// SIMATIC STEP 7 (V5.x) project DAYSILAUTOCLAVE
// CPU: CPU 315-2 PN/DP
// station: Hardware
// station: SLIO_CPU_015
// station: P_ADR_BUS
// program: S7 Program(1)
// program: 271220024

SYMBOL_TABLE
"AI-SENSOR-DATA"	DB 1	DB 1
"ORTAK_DATA"	DB 2	DB 2	// Ortak Veriler
"TIME_OTO_1_DB"	DB 5	SFB 4
"TIME_OTO_2_DB"	DB 6	SFB 4
"TIME_OTO_1_PROSES_DB"	DB 7	SFB 4
"TIME_OTO_2_PROSES_DB"	DB 8	SFB 4
"SURELER_DB"	DB 14	FB 3
"SAFETY_DB"	DB 15	FB 2
"KAZAN1_DATA"	DB 17	DB 17
"KAZAN2_DATA"	DB 18	DB 18	// KAZAN 2 BILGILERI
"JEN1_DATA"	DB 19	DB 19
"JEN2_DATA"	DB 20	DB 20
"JEN1_PID_DATA"	DB 21	DB 21
"JEN2_PID_DATA"	DB 22	DB 22
"KAZAN1_PID_DATA"	DB 23	DB 23	// KAZAN 1 PID BILGILERI
"KAZAN2_PID_DATA"	DB 24	DB 24	// KAZAN 2 PID BILGILERI
"JEN2_KONTROL_BLOGU_DB"	DB 51	FB 50
"JEN_1_PID_DB"	DB 69	FB 58
"JEN_2_PID_DB"	DB 70	FB 58
"OTOKLAV_1_DB"	DB 94	FB 94
"OTOKLAV_2_DB"	DB 95	FB 95
"FB98_DB"	DB 98	FB 98
"FB99_DB"	DB 99	FB 99
"HMI_DATA"	DB 100	DB 100	// Hmi arayuz verileri
"KAZAN_1_PID_DB"	DB 130	FB 58
"KAZAN_2_PID_DATA"	DB 231	FB 58
"MAINBLOCK"	FB 1	FB 1	// ANA PROGRAM BLOGU
"SAFETY"	FB 2	FB 2
"SURELER"	FB 3	FB 3
"TEST_BLOGU"	FB 5	FB 5
"KAZAN_ORTAK"	FB 20	FB 20
"KAZAN_PID_ORTAK"	FB 21	FB 21
"CONT_C"	FB 41	FB 41	// Continuous Control
"KAZAN_1_PID_KONTROL"	FB 47	FB 47
"KAZAN_2_PID_KONTROL"	FB 48	FB 48
"JEN1_PID_KONTROL"	FB 49	FB 49
"JEN2_PID_KONTROL"	FB 50	FB 50	// BUAHR JENERATÖR 2 PID
"TCONT_CP"	FB 58	FB 58	// temperature PID controller with pulse generator and self-tuning
"KAZAN_1_KONTROL"	FB 94	FB 94
"KAZAN_2_KONTROL"	FB 95	FB 95
"KAZAN1_KONTROL_BLOGU"	FB 96	FB 96
"KAZAN2_KONTROL_BLOGU"	FB 97	FB 97
"JEN1_KONTROL_BLOGU"	FB 98	FB 98
"JEN2_KONTROL_BLOGU"	FB 99	FB 99
"TIME_UNSCALE"	FC 1	FC 1
"S5TI_TIM"	FC 33	FC 33	// S5 Time to IEC Time
"SCALE"	FC 105	FC 105	// Scaling Values
"UNSCALE"	FC 106	FC 106	// Unscaling Values
"KAZAN1_ACIL_STOP"	I 0.0	BOOL	// Acil Stop
"KAZAN1_START"	I 0.1	BOOL	// Kazan 1 Start
"KAZAN1_TRANSFER"	I 0.2	BOOL	// Kazan 1 Buhar Transferi
"KAZAN1_BOSALTIM"	I 0.3	BOOL	// Kazan 1 Bosaltim
"KAZAN1_KAPAK_SW"	I 0.4	BOOL	// Kazan 1 Kapak Kapandi
"KAZAN2_ACIL_STOP"	I 0.5	BOOL	// Kazan 2 Acil Stop
"KAZAN2_START"	I 0.6	BOOL	// Kazan 2 Start
"KAZAN2_TRANSFER"	I 0.7	BOOL	// Kazan 2 Buhar Transferi
"KAZAN2_BOSALTIM"	I 1.0	BOOL	// Kazan 2 Bosaltim
"KAZAN2_KAPAK_SW"	I 1.1	BOOL	// Kazan 2 Kapak Kapandi
"JEN1_STOP"	I 1.2	BOOL	// Jenerator 1 Stop
"JEN1_START"	I 1.3	BOOL	// Jenerator 1 Start
"JEN2_STOP"	I 1.4	BOOL	// Jenerator 2 Stop
"JEN2_START"	I 1.5	BOOL	// Jenerator 2 Start
"MANUEL"	I 1.6	BOOL	// Manuel Mod
"OTOMATIK"	I 1.7	BOOL	// Otomatik Mod
"JEN2_MOTOR_CALISTI"	I 2.0	BOOL
"JEN_1_MIN_SU_SEVIYESI"	I 3.0	BOOL
"JEN_2_MIN_SU_SEVIYESI"	I 3.1	BOOL
"0.1 SN."	M 0.0	BOOL
"0.2 SN."	M 0.1	BOOL
"0.4 SN."	M 0.2	BOOL
"0.5 SN."	M 0.3	BOOL
"0.8 SN."	M 0.4	BOOL
"1.0 SN."	M 0.5	BOOL
"1.6 SN."	M 0.6	BOOL
"2.0 SN."	M 0.7	BOOL
"Oto_1_Proses_BASLADI"	M 20.0	BOOL
"Oto_2_Proses_Basladi"	M 20.1	BOOL
"JEN2_CALIS_SURESI_BASLA"	M 22.0	BOOL
"JEN2_CALISTI_RIS"	M 22.1	BOOL
"JEN1_CALIS_SURESI_BASLA"	M 23.0	BOOL
"JEN1_CALISTI_RIS"	M 23.1	BOOL
"Jen1_Guvenlik_set_reset"	M 25.0	BOOL
"Jen2_Guvenlik_Set_Reset"	M 26.0	BOOL
"OTO_1_BEKLEME_BASLADI"	M 27.0	BOOL
"OTO_2_BEKLEME_BASLADI"	M 27.1	BOOL
"KAZAN_1_PID_MAN_ON"	M 35.0	BOOL
"KAZAN_2_MAN_ON"	M 37.0	BOOL
"TEST_START"	M 40.0	BOOL
"TEST_STOP"	M 40.1	BOOL
"TEST_OUT"	M 40.2	BOOL
"ALWAYS OFF"	M 100.0	BOOL	// ALWAYS OFF
"ALWAYS ON"	M 100.1	BOOL	// ALWAYS ON
"SET2_ULASMADI_SR"	M 101.0	BOOL
"SET2_ULASMADI_RIS"	M 101.1	BOOL
"JEN2_TCONT_MAN_ON"	M 155.0	BOOL
"Jen2_Stop_Trigger"	M 200.0	BOOL
"Jen2_Stop_Ris"	M 200.1	BOOL
"Jen2_Stop_Set_Mem"	M 200.2	BOOL
"JEN2_STOP_SET_RESET"	M 201.0	BOOL
"Sicaklik Dustu"	M 201.1	BOOL
"Ris_Jen2_Sicaklik_Dustu"	M 201.2	BOOL
"Rising_Sogutma"	M 201.3	BOOL
"Falling_Sogutma"	M 201.4	BOOL
"JEN1_STOP_SET_RESET"	M 202.0	BOOL
"START"	M 700.1	BOOL
"PID_START"	M 700.2	BOOL
"BRULOR_START"	M 700.3	BOOL
"SICAKLIK_1_OK"	M 700.5	BOOL
"SICAKLIK_2_OK"	M 700.6	BOOL
"BURLOR_MOTOR_START"	M 700.7	BOOL
"STOP"	M 701.1	BOOL
"100_DERECE_RIS"	M 750.0	BOOL
"Jen2_Ris"	M 750.4	BOOL
"Jen1_Ris"	M 750.5	BOOL
"BOS"	M 1000.0	BOOL
"PID BLOCK"	OB 35	OB 35	// PID BLOCK
"ZAMANHATASI"	OB 80	OB 80	// ZAMAN HATASI
"GERILIMHATASI"	OB 81	OB 81	// BESLEME GERILIMI HATASI
"HATAUYARISI"	OB 82	OB 82	// HATA UYARISI
"TAKMACIKARMAHATASI"	OB 83	OB 83	// TAKMA ÇIKARMA UYARISI
"CPUHARDWAREERROR"	OB 84	OB 84	// CPU HARDWARE ERROR
"PROGRAMHATASI"	OB 85	OB 85	// PROGRAM YURUTME HATASI
"RACKHATASI"	OB 86	OB 86	// RACK HATASI
"HABERLESMEHATASI"	OB 87	OB 87	// HABERLESME HATASI,
"COMPLETE RESTART"	OB 100	OB 100	// Complete Restart
"RESTART"	OB 101	OB 101	// Restart
"COLD RESTART"	OB 102	OB 102	// Cold Restart
"PROGRAMMINGERROR"	OB 121	OB 121	// PROGRAMLAMA HATASI
"KAZAN1_YESIL_LAMBA"	Q 0.0	BOOL	// Kazan 1 Yesil Lamba
"KAZAN1_KIRMIZI_LAMBA"	Q 0.1	BOOL	// Kazan 1 Kirmizi Lamba
"KAZAN1_DUDUK"	Q 0.2	BOOL	// Kazan 1 Duduk
"KAZAN1_BOSALTIM_VALFI"	Q 0.3	BOOL	// Kazan 1 Buhar Bosaltim
"KAZAN1_TRANS_BUT_LAMBASI"	Q 0.4	BOOL	// Kazan 1 Transfer Lambasi
"KAZAN1_EMN_VALFI_BOS"	Q 0.5	BOOL	// Kazan  1 Emniyet vantili bosaltim valfi
"KAZAN2_YESIL_LAMBA"	Q 0.6	BOOL	// Kazan 2 Yesil Lamba
"KAZAN2_KIRMIZI_LAMBA"	Q 0.7	BOOL	// Kazan 2 Kirmizi Lamba
"KAZAN2_DUDUK"	Q 1.0	BOOL	// Kazan 2 Duduk
"KAZAN2_BOSALTIM_VALFI"	Q 1.1	BOOL	// Kazan 2 Buhar Bosaltim
"KAZAN2_TRANS_BUT_LAMBASI"	Q 1.2	BOOL	// Kazan 2 Transfer Lambasi
"KAZAN2_EMN_VALFI_BOS"	Q 1.3	BOOL	// Kazan Emniyet vantili bosaltim valfi
"JEN_1_HAT_VANASI"	Q 1.4	BOOL
"JEN_1_PANO_STOP_LAMBASI"	Q 1.5	BOOL
"JEN_1_PANO_START_LAMBASI"	Q 1.6	BOOL
"JEN_2_HAT_VANASI"	Q 1.7	BOOL
"JEN_2_PANO_STOP_LAMBASI"	Q 2.0	BOOL
"JEN_2_PANO_START_LAMBASI"	Q 2.1	BOOL
"PANO_OTO_MAN_BUTON_LAMBA"	Q 2.2	BOOL
"PANO_ALARM"	Q 2.3	BOOL
"JEN_1_BRULOR"	Q 2.4	BOOL
"JEN_1_POMPA"	Q 2.5	BOOL
"JEN_2_BRULOR_OUT"	Q 2.6	BOOL
"JEN_2_SU_POM_OUT"	Q 2.7	BOOL
"TON"	SFB 4	SFB 4	// Generate an On Delay
"delay_300ms_1"	T 8	TIMER
"500ms_delay1"	T 10	TIMER
"1s Delay"	T 11	TIMER
"Pisim_Suresi"	T 12	TIMER
"500ms_delay"	T 13	TIMER
"s_offt_7s_delay"	T 14	TIMER
"tm_adim1_pid_basla_delay"	T 16	TIMER
"500ms_delay_kazan_2"	T 20	TIMER
"1ms_delay_kazan_2"	T 21	TIMER
"kazan_2_pisirme_delay"	T 22	TIMER
"kazan_2_500ms_delay"	T 23	TIMER
"kazan_2_7s_delay"	T 24	TIMER
"Delay_500ms_Jen2"	T 30	TIMER
"DELAY_1S_JEN_HATA"	T 33	TIMER
"DELAY_300MS"	T 42	TIMER
"DELAY_500MS_1"	T 43	TIMER
"DELAY_5S_pompa"	T 44	TIMER
"OTO_2_DELAY_BITIS"	T 50	TIMER
"OTO_1_DELAY_PISIM_BITTI"	T 51	TIMER
"DELAY_ADIM5_BEKLE"	T 52	TIMER
"DELAY_ADIM5_BEKLE2"	T 53	TIMER
"TIM_SET2_ULASMADI"	T 57	TIMER
"TEST BLOGU VAT"	VAT 1	
"JEN2_MONITOR"	VAT 2	
"KAZAN-1-MONITOR"	VAT 3	
"KAZAN-2-MONITOR"	VAT 4	
"JEN1_MONITOR"	VAT 5	
"deneme"	VAT 6	
END_SYMBOL_TABLE

FUNCTION_BLOCK "MAINBLOCK"	// FB 1
VERSION : 0.1
BEGIN
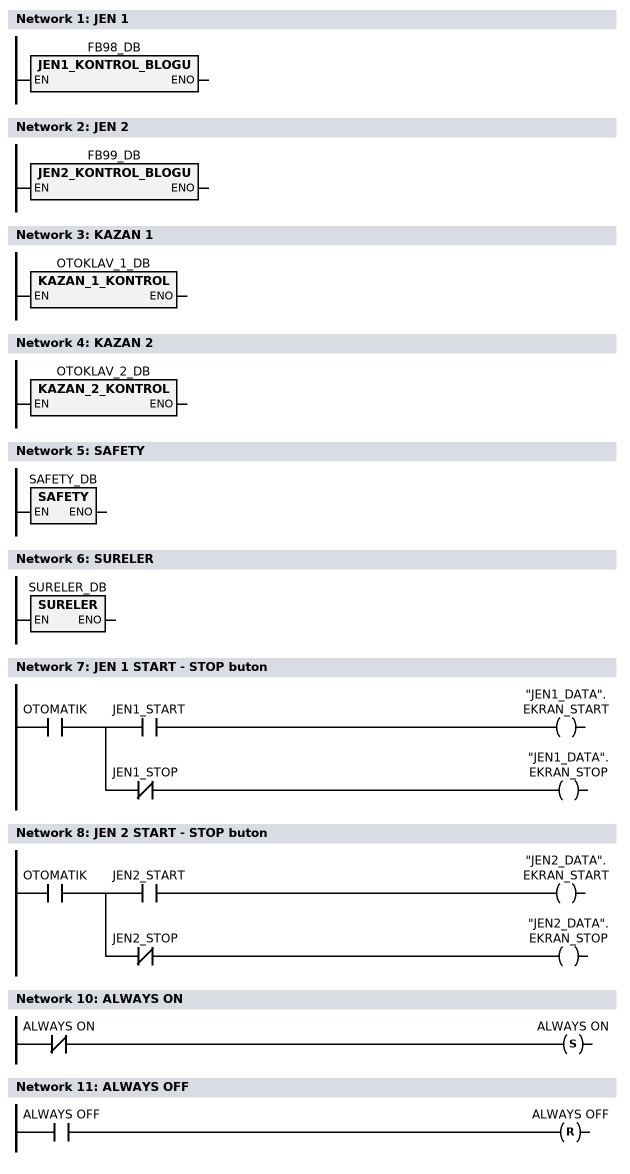
NETWORK
TITLE = JEN 1
      CALL  "JEN1_KONTROL_BLOGU" , "FB98_DB";
      NOP   0;
NETWORK
TITLE = JEN 2
      CALL  "JEN2_KONTROL_BLOGU" , "FB99_DB";
      NOP   0;
NETWORK
TITLE = KAZAN 1
      CALL  "KAZAN_1_KONTROL" , "OTOKLAV_1_DB";
      NOP   0;
NETWORK
TITLE = KAZAN 2
      CALL  "KAZAN_2_KONTROL" , "OTOKLAV_2_DB";
      NOP   0;
NETWORK
TITLE = SAFETY
      CALL  "SAFETY" , "SAFETY_DB";
      NOP   0;
NETWORK
TITLE = SURELER
      CALL  "SURELER" , "SURELER_DB";
      NOP   0;
NETWORK
TITLE = JEN 1 START - STOP buton
      A     "OTOMATIK";
      =     L 0.0;
      A     L 0.0;
      A     "JEN1_START";
      =     "JEN1_DATA".EKRAN_START;
      A     L 0.0;
      AN    "JEN1_STOP";
      =     "JEN1_DATA".EKRAN_STOP;
NETWORK
TITLE = JEN 2 START - STOP buton
      A     "OTOMATIK";
      =     L 0.0;
      A     L 0.0;
      A     "JEN2_START";
      =     "JEN2_DATA".EKRAN_START;
      A     L 0.0;
      AN    "JEN2_STOP";
      =     "JEN2_DATA".EKRAN_STOP;
NETWORK
TITLE =
NETWORK
TITLE = ALWAYS ON
      AN    "ALWAYS ON";
      S     "ALWAYS ON";
NETWORK
TITLE = ALWAYS OFF
      A     "ALWAYS OFF";
      R     "ALWAYS OFF";
NETWORK
TITLE =
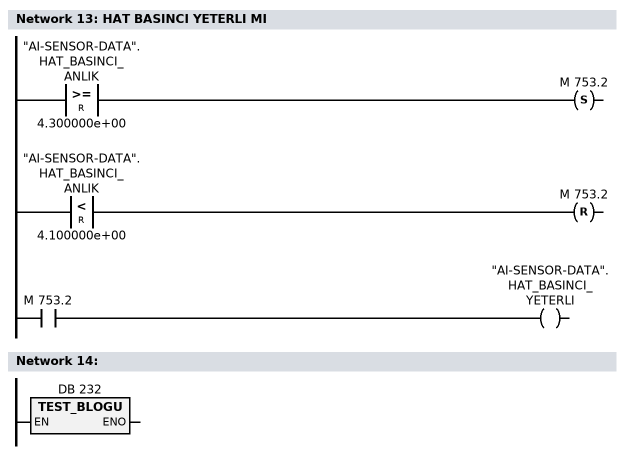
NETWORK
TITLE = HAT BASINCI YETERLI MI
      A(;
      L     "AI-SENSOR-DATA".HAT_BASINCI_ANLIK;
      L     4.300000e+00;
      >=R;
      );
      S     M 753.2;
      A(;
      L     "AI-SENSOR-DATA".HAT_BASINCI_ANLIK;
      L     4.100000e+00;
      <R;
      );
      R     M 753.2;
      A     M 753.2;
      =     "AI-SENSOR-DATA".HAT_BASINCI_YETERLI;
NETWORK
TITLE =
      CALL  "TEST_BLOGU" , DB 232;
      NOP   0;
END_FUNCTION_BLOCK

FUNCTION_BLOCK "SAFETY"	// FB 2
VERSION : 0.1
BEGIN
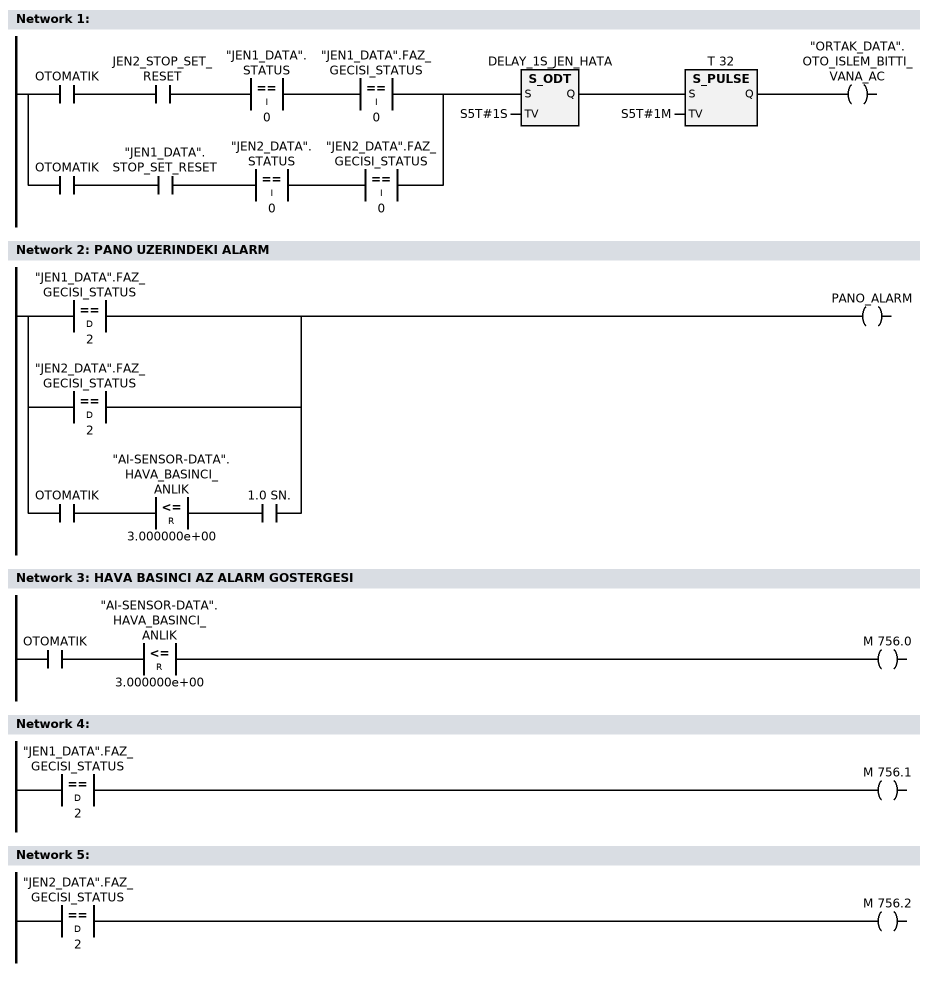
NETWORK
TITLE =
      A(;
      A(;
      A     "OTOMATIK";
      A     "JEN2_STOP_SET_RESET";
      A(;
      L     "JEN1_DATA".STATUS;
      L     0;
      ==I;
      );
      A(;
      L     "JEN1_DATA".FAZ_GECISI_STATUS;
      L     0;
      ==I;
      );
      O;
      A     "OTOMATIK";
      A     "JEN1_DATA".STOP_SET_RESET;
      A(;
      L     "JEN2_DATA".STATUS;
      L     0;
      ==I;
      );
      A(;
      L     "JEN2_DATA".FAZ_GECISI_STATUS;
      L     0;
      ==I;
      );
      );
      L     S5T#1S;
      SD    "DELAY_1S_JEN_HATA";
      NOP   0;
      NOP   0;
      NOP   0;
      A     "DELAY_1S_JEN_HATA";
      );
      L     S5T#1M;
      SP    T 32;
      NOP   0;
      NOP   0;
      NOP   0;
      A     T 32;
      =     "ORTAK_DATA".OTO_ISLEM_BITTI_VANA_AC;
NETWORK
TITLE = PANO UZERINDEKI ALARM 
//JENERATORDE MINIMUM SU SEVIYESINE DUSERSE PANO UZERINDEKI ALARMI CALISTIR
      O(;
      L     "JEN1_DATA".FAZ_GECISI_STATUS;
      L     2;
      ==D;
      );
      O(;
      L     "JEN2_DATA".FAZ_GECISI_STATUS;
      L     2;
      ==D;
      );
      O;
      A     "OTOMATIK";
      A(;
      L     "AI-SENSOR-DATA".HAVA_BASINCI_ANLIK;
      L     3.000000e+00;
      <=R;
      );
      A     "1.0 SN.";
      =     "PANO_ALARM";
NETWORK
TITLE = HAVA BASINCI AZ ALARM GOSTERGESI
      A     "OTOMATIK";
      A(;
      L     "AI-SENSOR-DATA".HAVA_BASINCI_ANLIK;
      L     3.000000e+00;
      <=R;
      );
      =     M 756.0;
NETWORK
TITLE =
      L     "JEN1_DATA".FAZ_GECISI_STATUS;
      L     2;
      ==D;
      =     M 756.1;
NETWORK
TITLE =
      L     "JEN2_DATA".FAZ_GECISI_STATUS;
      L     2;
      ==D;
      =     M 756.2;
END_FUNCTION_BLOCK

FUNCTION_BLOCK "SURELER"	// FB 3
VERSION : 0.1
BEGIN
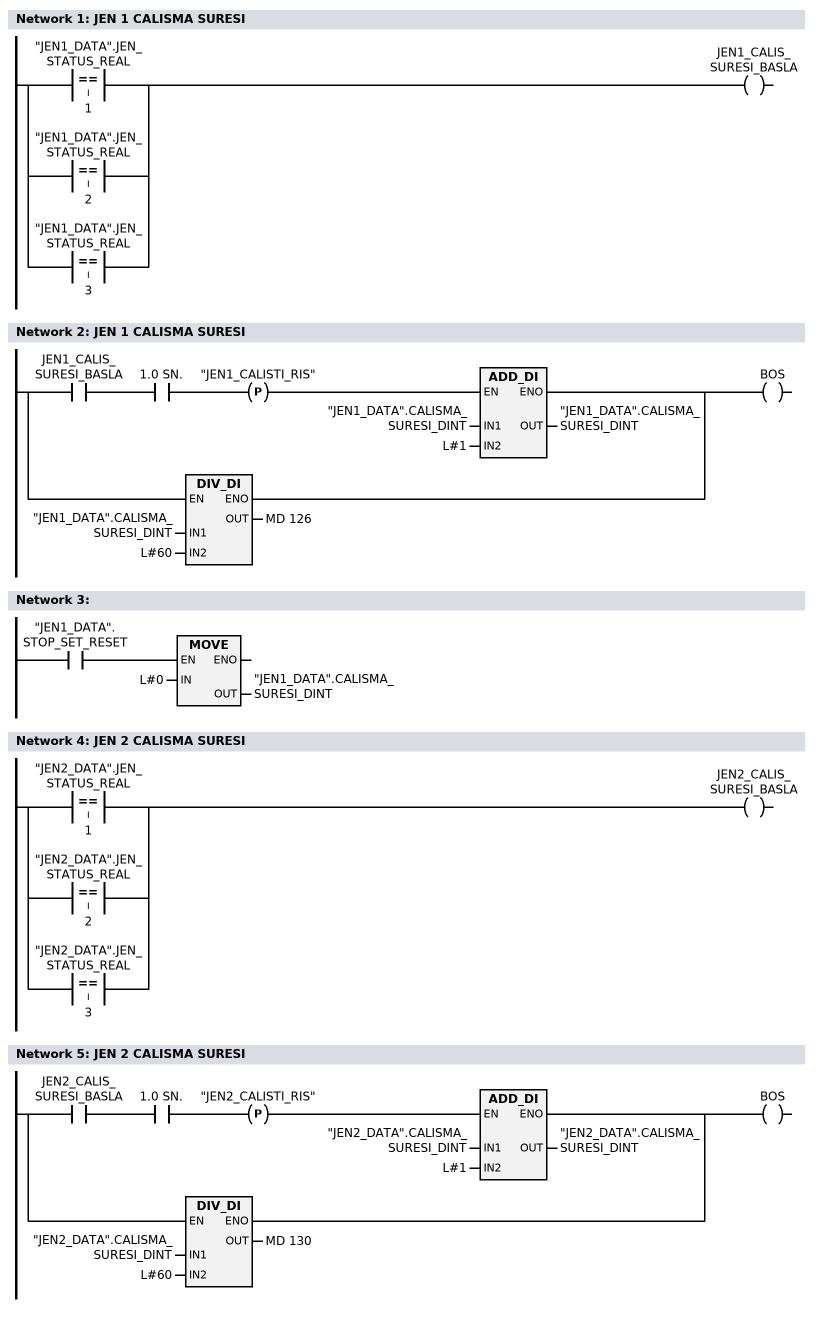
NETWORK
TITLE = JEN 1 CALISMA SURESI
      O(;
      L     "JEN1_DATA".JEN_STATUS_REAL;
      L     1;
      ==I;
      );
      O(;
      L     "JEN1_DATA".JEN_STATUS_REAL;
      L     2;
      ==I;
      );
      O(;
      L     "JEN1_DATA".JEN_STATUS_REAL;
      L     3;
      ==I;
      );
      =     "JEN1_CALIS_SURESI_BASLA";
NETWORK
TITLE = JEN 1 CALISMA SURESI
      O(;
      A     "JEN1_CALIS_SURESI_BASLA";
      A     "1.0 SN.";
      FP    "JEN1_CALISTI_RIS";
      JNB   _001;
      L     "JEN1_DATA".CALISMA_SURESI_DINT;
      L     L#1;
      +D;
      T     "JEN1_DATA".CALISMA_SURESI_DINT;
      AN    OV;
      SAVE;
      CLR;
_001: A     BR;
      );
      O(;
      L     "JEN1_DATA".CALISMA_SURESI_DINT;
      L     L#60;
      /D;
      T     MD 126;
      AN    OV;
      SAVE;
      CLR;
      A     BR;
      );
      =     "BOS";
NETWORK
TITLE =
      A     "JEN1_DATA".STOP_SET_RESET;
      JNB   _002;
      L     L#0;
      T     "JEN1_DATA".CALISMA_SURESI_DINT;
_002: NOP   0;
NETWORK
TITLE = JEN 2 CALISMA SURESI
      O(;
      L     "JEN2_DATA".JEN_STATUS_REAL;
      L     1;
      ==I;
      );
      O(;
      L     "JEN2_DATA".JEN_STATUS_REAL;
      L     2;
      ==I;
      );
      O(;
      L     "JEN2_DATA".JEN_STATUS_REAL;
      L     3;
      ==I;
      );
      =     "JEN2_CALIS_SURESI_BASLA";
NETWORK
TITLE = JEN 2 CALISMA SURESI
      O(;
      A     "JEN2_CALIS_SURESI_BASLA";
      A     "1.0 SN.";
      FP    "JEN2_CALISTI_RIS";
      JNB   _003;
      L     "JEN2_DATA".CALISMA_SURESI_DINT;
      L     L#1;
      +D;
      T     "JEN2_DATA".CALISMA_SURESI_DINT;
      AN    OV;
      SAVE;
      CLR;
_003: A     BR;
      );
      O(;
      L     "JEN2_DATA".CALISMA_SURESI_DINT;
      L     L#60;
      /D;
      T     MD 130;
      AN    OV;
      SAVE;
      CLR;
      A     BR;
      );
      =     "BOS";
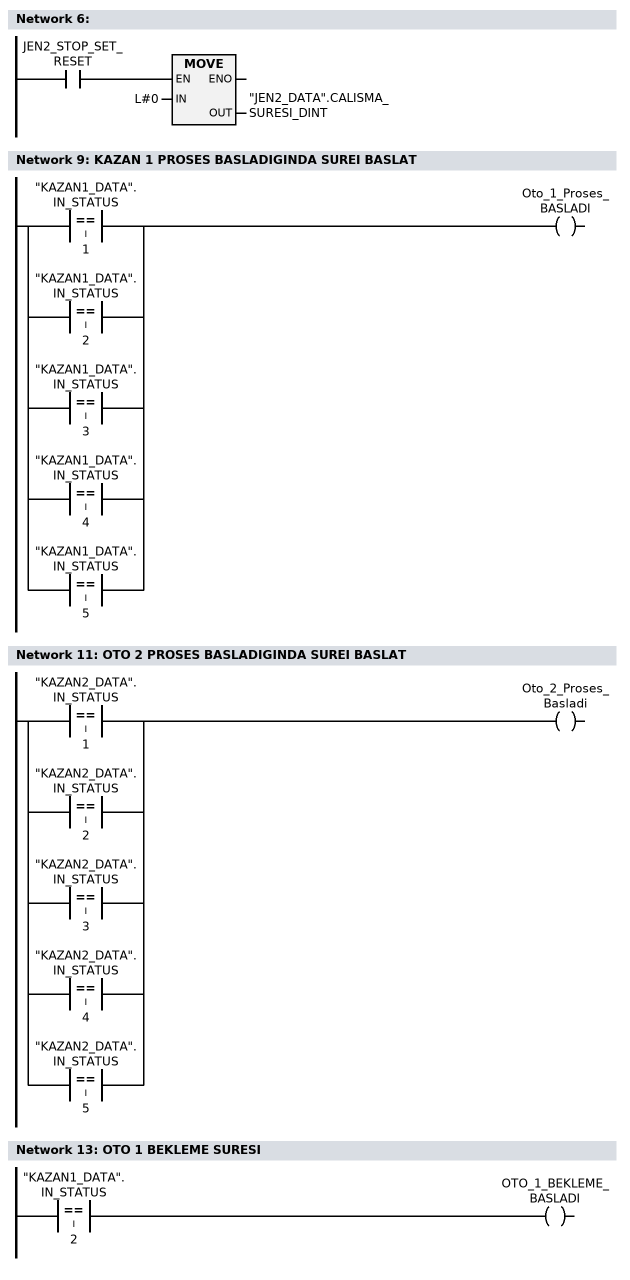
NETWORK
TITLE =
      A     "JEN2_STOP_SET_RESET";
      JNB   _004;
      L     L#0;
      T     "JEN2_DATA".CALISMA_SURESI_DINT;
_004: NOP   0;
NETWORK
TITLE = OTOKLAV 1 PISIM GECEN SURE
      O(;
      A(;
      A     "KAZAN1_DATA".O_PISIM_BASLADI;
      =     L 0.0;
      BLD   103;
      BLD   9;
      =     L 5.0;
      CDB;
      OPN   DI 5;
      TAR2  LD 1;
      A     L 0.0;
      =     DIX 0.0;
      L     L#82800000;
      T     DID 2;
      LAR2  P#DBX 0.0;
      UC    "TON";
      LAR2  LD 1;
      L     DID 8;
      OPN   DI 17;
      T     DID 42;
      OPN   DI 5;
      CDB;
      BLD   10;
      A     BR;
      );
      JNB   _005;
      CALL  "TIME_UNSCALE" (
           iTimeET                  := "KAZAN1_DATA".PISIM_GECEN_SURE_TIME,
           iIstenileSure            := "KAZAN1_DATA".IN_PISIM_SURESI,
           oOUT                     := "KAZAN1_DATA".PISIM_GECEN_SURE_DINT);
_005: A     BR;
      );
      O(;
      L     "KAZAN1_DATA".PISIM_GECEN_SURE_DINT;
      L     60;
      /D;
      T     MD 118;
      AN    OV;
      SAVE;
      CLR;
      A     BR;
      );
      =     "BOS";
NETWORK
TITLE = OTOKLAV 2 PISIM GECEN SURE
      O(;
      A(;
      A     "KAZAN2_DATA".O_PISIM_BASLADI;
      =     L 0.0;
      BLD   103;
      BLD   9;
      =     L 5.0;
      CDB;
      OPN   DI 6;
      TAR2  LD 1;
      A     L 0.0;
      =     DIX 0.0;
      L     L#82800000;
      T     DID 2;
      LAR2  P#DBX 0.0;
      UC    "TON";
      LAR2  LD 1;
      L     DID 8;
      OPN   DI 18;
      T     DID 42;
      OPN   DI 6;
      CDB;
      BLD   10;
      A     BR;
      );
      JNB   _006;
      CALL  "TIME_UNSCALE" (
           iTimeET                  := "KAZAN2_DATA".PISIM_GECEN_SURE_TIME,
           iIstenileSure            := "KAZAN2_DATA".IN_PISIM_SURESI,
           oOUT                     := "KAZAN2_DATA".PISIM_GECEN_SURE_DINT);
_006: A     BR;
      );
      O(;
      L     "KAZAN2_DATA".PISIM_GECEN_SURE_DINT;
      L     60;
      /D;
      T     MD 122;
      AN    OV;
      SAVE;
      CLR;
      A     BR;
      );
      =     "BOS";
NETWORK
TITLE = KAZAN 1 PROSES BASLADIGINDA SUREI BASLAT
      O(;
      L     "KAZAN1_DATA".IN_STATUS;
      L     1;
      ==I;
      );
      O(;
      L     "KAZAN1_DATA".IN_STATUS;
      L     2;
      ==I;
      );
      O(;
      L     "KAZAN1_DATA".IN_STATUS;
      L     3;
      ==I;
      );
      O(;
      L     "KAZAN1_DATA".IN_STATUS;
      L     4;
      ==I;
      );
      O(;
      L     "KAZAN1_DATA".IN_STATUS;
      L     5;
      ==I;
      );
      =     "Oto_1_Proses_BASLADI";
NETWORK
TITLE = OTOKLAV 1 PROSES SURESI
      O(;
      A(;
      A     "Oto_1_Proses_BASLADI";
      =     L 0.0;
      BLD   103;
      BLD   9;
      =     L 5.0;
      CDB;
      OPN   DI 7;
      TAR2  LD 1;
      A     L 0.0;
      =     DIX 0.0;
      L     L#82800000;
      T     DID 2;
      LAR2  P#DBX 0.0;
      UC    "TON";
      LAR2  LD 1;
      L     DID 8;
      OPN   DI 17;
      T     DID 50;
      OPN   DI 7;
      CDB;
      BLD   10;
      A     BR;
      );
      JNB   _007;
      L     "KAZAN1_DATA".PROSES_SURESI_TIME;
      L     1000;
      /D;
      T     "KAZAN1_DATA".PROSES_SURESI_DINT;
      AN    OV;
      SAVE;
      CLR;
_007: A     BR;
      );
      O(;
      L     "KAZAN1_DATA".PROSES_SURESI_DINT;
      L     60;
      /D;
      T     MD 110;
      AN    OV;
      SAVE;
      CLR;
      A     BR;
      );
      =     "BOS";
NETWORK
TITLE = OTO 2 PROSES BASLADIGINDA SUREI BASLAT
      O(;
      L     "KAZAN2_DATA".IN_STATUS;
      L     1;
      ==I;
      );
      O(;
      L     "KAZAN2_DATA".IN_STATUS;
      L     2;
      ==I;
      );
      O(;
      L     "KAZAN2_DATA".IN_STATUS;
      L     3;
      ==I;
      );
      O(;
      L     "KAZAN2_DATA".IN_STATUS;
      L     4;
      ==I;
      );
      O(;
      L     "KAZAN2_DATA".IN_STATUS;
      L     5;
      ==I;
      );
      =     "Oto_2_Proses_Basladi";
NETWORK
TITLE = OTO 2 PROSES_SURESI
      O(;
      A(;
      A     "Oto_2_Proses_Basladi";
      =     L 0.0;
      BLD   103;
      BLD   9;
      =     L 5.0;
      CDB;
      OPN   DI 8;
      TAR2  LD 1;
      A     L 0.0;
      =     DIX 0.0;
      L     L#82800000;
      T     DID 2;
      LAR2  P#DBX 0.0;
      UC    "TON";
      LAR2  LD 1;
      L     DID 8;
      OPN   DI 18;
      T     DID 50;
      OPN   DI 8;
      CDB;
      BLD   10;
      A     BR;
      );
      JNB   _008;
      L     "KAZAN2_DATA".PROSES_SURESI_TIM;
      L     1000;
      /D;
      T     "KAZAN2_DATA".PROSES_SURESI_DINT;
      AN    OV;
      SAVE;
      CLR;
_008: A     BR;
      );
      O(;
      L     "KAZAN2_DATA".PROSES_SURESI_DINT;
      L     60;
      /D;
      T     MD 114;
      AN    OV;
      SAVE;
      CLR;
      A     BR;
      );
      =     "BOS";
NETWORK
TITLE = OTO 1 BEKLEME SURESI
      L     "KAZAN1_DATA".IN_STATUS;
      L     2;
      ==I;
      =     "OTO_1_BEKLEME_BASLADI";
NETWORK
TITLE = OTO 1 BEKLEME SURESI
      A(;
      A     "OTO_1_BEKLEME_BASLADI";
      =     L 0.0;
      BLD   103;
      BLD   9;
      =     L 5.0;
      CDB;
      OPN   DI 9;
      TAR2  LD 1;
      A     L 0.0;
      =     DIX 0.0;
      L     L#82800000;
      T     DID 2;
      LAR2  P#DBX 0.0;
      UC    "TON";
      LAR2  LD 1;
      L     DID 8;
      OPN   DI 17;
      T     DID 58;
      OPN   DI 9;
      CDB;
      BLD   10;
      A     BR;
      );
      JNB   _009;
      L     "KAZAN1_DATA".BEKLEME_SURESI_TIME;
      L     1000;
      /D;
      T     "KAZAN1_DATA".BEKLEME_SURESI_DINT;
_009: NOP   0;
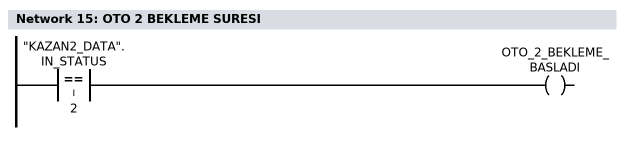
NETWORK
TITLE = OTO 2 BEKLEME SURESI
      L     "KAZAN2_DATA".IN_STATUS;
      L     2;
      ==I;
      =     "OTO_2_BEKLEME_BASLADI";
NETWORK
TITLE = OTO 2 BEKLEME SURESI
      A(;
      A     "OTO_2_BEKLEME_BASLADI";
      =     L 0.0;
      BLD   103;
      BLD   9;
      =     L 5.0;
      CDB;
      OPN   DI 10;
      TAR2  LD 1;
      A     L 0.0;
      =     DIX 0.0;
      L     L#82800000;
      T     DID 2;
      LAR2  P#DBX 0.0;
      UC    "TON";
      LAR2  LD 1;
      L     DID 8;
      OPN   DI 18;
      T     DID 58;
      OPN   DI 10;
      CDB;
      BLD   10;
      A     BR;
      );
      JNB   _00a;
      L     "KAZAN2_DATA".BEKLEME_SURESI_TIME;
      L     1000;
      /D;
      T     "KAZAN2_DATA".BEKLEME_SURESI_DINT;
_00a: NOP   0;
END_FUNCTION_BLOCK

FUNCTION_BLOCK "TEST_BLOGU"	// FB 5
VERSION : 0.1
BEGIN
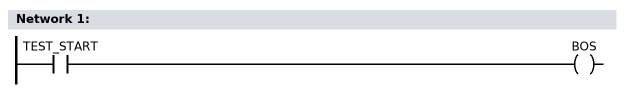
NETWORK
TITLE =
      A     "TEST_START";
      =     "BOS";
END_FUNCTION_BLOCK

FUNCTION_BLOCK "KAZAN_ORTAK"	// FB 20
//0 - baslama kriterleri
//1 - pid baslasin
//
VERSION : 0.1
VAR_INPUT
  IN_ACIL_STOP : BOOL ;
  IN_START : BOOL ;
  IN_TRANSFER : BOOL ;
  IN_BOSALTIM : BOOL ;
  IN_KAPAK : BOOL ;
  IN_JEN1_OK : BOOL ;
  IN_JEN2_OK : BOOL ;
  IN_JENS_OK : BOOL ;
  IN_TRANSFERE_HAZIR : BOOL ;
  IN_PISIM_SURESI : S5TIME ;
  IN_SCALE_BASINC_PER : INT ;
  IN_SET_BASINC : REAL ;
  IN_DIGER_KAZAN_BASINCI : REAL ;
  IN_TIMER_500MS : TIMER ;
  IN_TIMER_1S : TIMER ;
  IN_TIMER_PISIRME : TIMER ;
  IN_TIMER_500MS_2 : TIMER ;
  IN_TIMER_7S : TIMER ;
  IN_SCALE_HI_LIM : REAL ;
  IN_SCALE_LO_LIM : REAL ;
  IN_SCALE_SICAKLIK_HI_LIM : REAL ;
  IN_SCALE_SICAKLIK_LO_LIM : REAL ;
  IN_SCALE_SICAKLIK_PER : INT ;
  IN_DIGER_KAZAN_BOSALTIMD : BOOL ;
  IN_TRANSFER_BASLADI : BOOL ;
  IN_PISIM_SURESI_TIME_DB : BLOCK_DB ;
  IN_DIG_KAZAN_PROSES_BAS : BOOL ;
  IN_JEN_DURDU : BOOL ;
  IN_JEN_DURDUR_PID_MAN : REAL ;
  IN_DELAY_BITISI_BEKLE : TIMER ;
  IN_DELAY_BIRAZ_BEKLE : TIMER ;
END_VAR
VAR_OUTPUT
  O_YESIL_LAM : BOOL ;
  O_KIRMIZI_LAM : BOOL ;
  O_DUDUK : BOOL ;
  O_BOSALTIM_VALFI : BOOL ;
  O_PID_MAN_ON : BOOL ;
  O_PID_MAN : REAL ;
  O_TRANSFER_YAPILIYOR : BOOL ;
  O_SCALE_BASINC_RET_VAL : WORD ;
  O_SCALE_BASINC_OUT : REAL ;
  O_EMNIYET_VALFI : BOOL ;
  O_TRANSFERE_HAZIR : BOOL ;
  O_SCALE_SICAKLIK_RET_VAL : WORD ;
  O_SCALE_SICAKLIK_OUT : REAL ;
  O_TRANSFER_ET_LAMBASI : BOOL ;
  O_PROSES_BASLADI : BOOL ;
  O_KAZAN_BOSALTIMDA : BOOL ;
  O_PISIM_BASLADI : BOOL ;
END_VAR
VAR_IN_OUT
  STATUS : INT ;
END_VAR
VAR
  ST_STATUS : INT ;
  ST_OUT_BOSALTIM_MEM : BOOL ;
  ST_OUT_PID_MAN_ON : BOOL ;
  ST_OUT_PID_MAN : REAL ;
  st_ris_pid_zero : BOOL ;
  st_scale_hi_lim : REAL  := 1.000000e+001;
  st_scale_lo_lim : REAL ;
  st_basinc_ok_sure_basla : BOOL ;
  st_tolerans_mul : REAL ;
  st_toleransli_basinc : REAL ;
  st_adim4_bosaltim_valfi : BOOL ;
  st_OUT_adim4_emnyet_val : BOOL ;
  st_pid_basla : BOOL ;
  st_bosalti_valfi_acil : BOOL ;
  st_scale_basinc_ret_val : WORD ;
  st_scale_basinc_out : REAL ;
  st_scale_sicaklik_ret_va : WORD ;
  st_scale_sicaklik_out : REAL ;
  ST_PROSES_BASLADI : BOOL ;
  ST_KAZAN_BOSALTIMDA : BOOL ;
  ST_BOS : BOOL ;
  ST_SET_ADD_BASINC_02 : REAL ;
  ST_GECEN_PISIM_SURESI : TIME ;
  st_5_bar_ustu : BOOL ;
  st_5_bar_alti : BOOL ;
  st_5_bar_guvenlik_SR : BOOL ;
  st_5_bar_guvenlik_mem : BOOL ;
END_VAR
BEGIN
NETWORK
TITLE = BASLANGIC SARTLARI
      A(;
      A(;
      A     "ALWAYS OFF";
      =     L 0.0;
      BLD   103;
      CALL  "SCALE" (
           $1                       := #IN_SCALE_BASINC_PER,
           $2                       := #IN_SCALE_HI_LIM,
           $3                       := #IN_SCALE_LO_LIM,
           $4                       := L 0.0,
           $5                       := #st_scale_basinc_ret_val,
           $6                       := #st_scale_basinc_out);
      A     BR;
      );
      JNB   _001;
      L     #st_scale_basinc_ret_val;
      T     #O_SCALE_BASINC_RET_VAL;
      SET;
      SAVE;
      CLR;
_001: A     BR;
      );
      JNB   _002;
      L     #st_scale_basinc_out;
      T     #O_SCALE_BASINC_OUT;
_002: NOP   0;
NETWORK
TITLE =
      A(;
      A(;
      A     "ALWAYS OFF";
      =     L 0.0;
      BLD   103;
      CALL  "SCALE" (
           $1                       := #IN_SCALE_SICAKLIK_PER,
           $2                       := #IN_SCALE_SICAKLIK_HI_LIM,
           $3                       := #IN_SCALE_SICAKLIK_LO_LIM,
           $4                       := L 0.0,
           $5                       := #st_scale_sicaklik_ret_va,
           $6                       := #st_scale_sicaklik_out);
      A     BR;
      );
      JNB   _003;
      L     #st_scale_sicaklik_ret_va;
      T     #O_SCALE_SICAKLIK_RET_VAL;
      SET;
      SAVE;
      CLR;
_003: A     BR;
      );
      JNB   _004;
      L     #st_scale_sicaklik_out;
      T     #O_SCALE_SICAKLIK_OUT;
_004: NOP   0;
NETWORK
TITLE = START
      A(;
      A     "OTOMATIK";
      A     #IN_ACIL_STOP;
      A     "AI-SENSOR-DATA".HAT_BASINCI_YETERLI;
      L     S5T#200MS;
      T     LD 0;
      TAK;
      T     LD 4;
      L     #IN_TIMER_500MS;
      T     LW 8;
      L     LD 4;
      L     LD 0;
      SD    T [LW 8];
      NOP   0;
      NOP   0;
      NOP   0;
      T     LD 0;
      TAK;
      T     LD 4;
      L     #IN_TIMER_500MS;
      T     LW 8;
      L     LD 4;
      L     LD 0;
      A     T [LW 8];
      );
      A     #IN_KAPAK;
      A     #IN_START;
      A(;
      L     #STATUS;
      L     0;
      ==I;
      );
      JNB   _005;
      L     1;
      T     #STATUS;
      SET;
      SAVE;
      CLR;
_005: A     BR;
      S     #ST_PROSES_BASLADI;
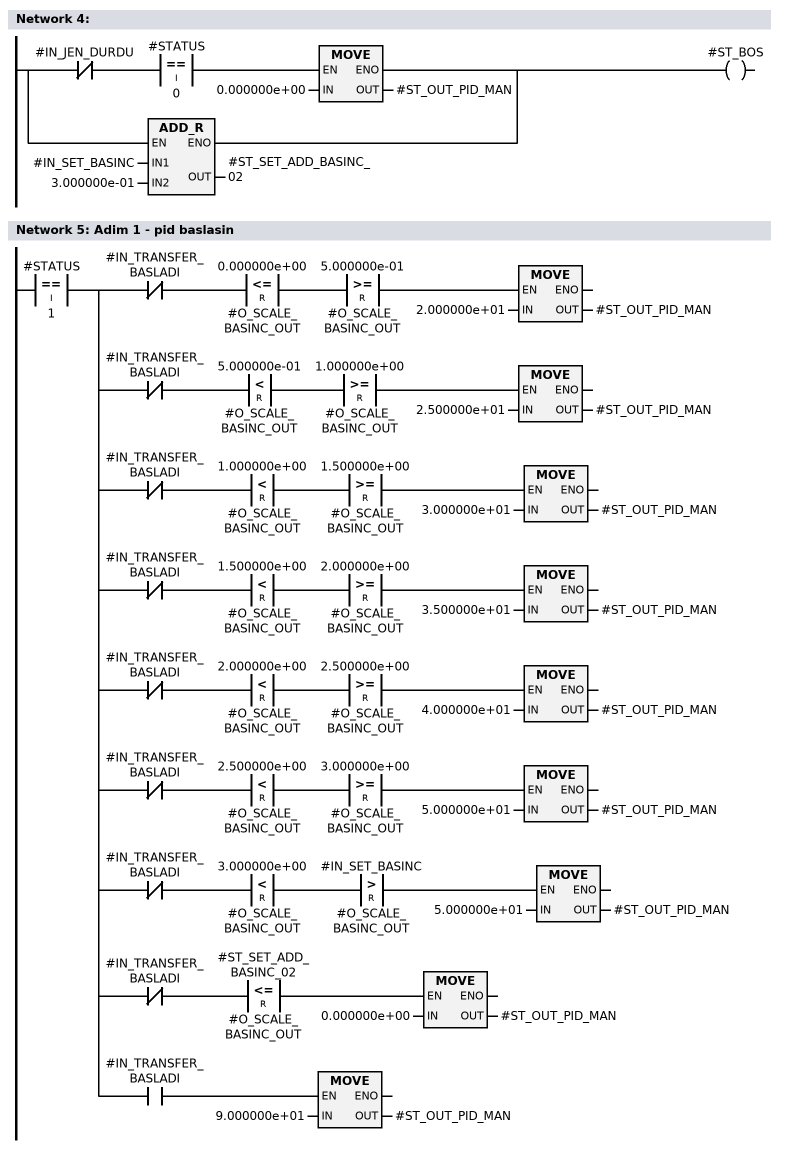
NETWORK
TITLE =
//1-Baslangicta vakum olmamasi icin bosaltim valfini ac
//Valf Normalde acik gibi dusundum
//2-Oransal valfi kapali tut
      O(;
      AN    #IN_JEN_DURDU;
      A(;
      L     #STATUS;
      L     0;
      ==I;
      );
      JNB   _006;
      L     0.000000e+00;
      T     #ST_OUT_PID_MAN;
      SET;
      SAVE;
      CLR;
_006: A     BR;
      );
      O(;
      L     #IN_SET_BASINC;
      L     3.000000e-01;
      +R;
      T     #ST_SET_ADD_BASINC_02;
      AN    OV;
      SAVE;
      CLR;
      A     BR;
      );
      =     #ST_BOS;
NETWORK
TITLE = Adim 1 - pid baslasin
      L     #STATUS;
      L     1;
      ==I;
      =     L 0.0;
      A     L 0.0;
      AN    #IN_TRANSFER_BASLADI;
      A(;
      L     0.000000e+00;
      L     #O_SCALE_BASINC_OUT;
      <=R;
      );
      A(;
      L     5.000000e-01;
      L     #O_SCALE_BASINC_OUT;
      >=R;
      );
      JNB   _007;
      L     2.000000e+01;
      T     #ST_OUT_PID_MAN;
_007: NOP   0;
      A     L 0.0;
      AN    #IN_TRANSFER_BASLADI;
      A(;
      L     5.000000e-01;
      L     #O_SCALE_BASINC_OUT;
      <R;
      );
      A(;
      L     1.000000e+00;
      L     #O_SCALE_BASINC_OUT;
      >=R;
      );
      JNB   _008;
      L     2.500000e+01;
      T     #ST_OUT_PID_MAN;
_008: NOP   0;
      A     L 0.0;
      AN    #IN_TRANSFER_BASLADI;
      A(;
      L     1.000000e+00;
      L     #O_SCALE_BASINC_OUT;
      <R;
      );
      A(;
      L     1.500000e+00;
      L     #O_SCALE_BASINC_OUT;
      >=R;
      );
      JNB   _009;
      L     3.000000e+01;
      T     #ST_OUT_PID_MAN;
_009: NOP   0;
      A     L 0.0;
      AN    #IN_TRANSFER_BASLADI;
      A(;
      L     1.500000e+00;
      L     #O_SCALE_BASINC_OUT;
      <R;
      );
      A(;
      L     2.000000e+00;
      L     #O_SCALE_BASINC_OUT;
      >=R;
      );
      JNB   _00a;
      L     3.500000e+01;
      T     #ST_OUT_PID_MAN;
_00a: NOP   0;
      A     L 0.0;
      AN    #IN_TRANSFER_BASLADI;
      A(;
      L     2.000000e+00;
      L     #O_SCALE_BASINC_OUT;
      <R;
      );
      A(;
      L     2.500000e+00;
      L     #O_SCALE_BASINC_OUT;
      >=R;
      );
      JNB   _00b;
      L     4.000000e+01;
      T     #ST_OUT_PID_MAN;
_00b: NOP   0;
      A     L 0.0;
      AN    #IN_TRANSFER_BASLADI;
      A(;
      L     2.500000e+00;
      L     #O_SCALE_BASINC_OUT;
      <R;
      );
      A(;
      L     3.000000e+00;
      L     #O_SCALE_BASINC_OUT;
      >=R;
      );
      JNB   _00c;
      L     5.000000e+01;
      T     #ST_OUT_PID_MAN;
_00c: NOP   0;
      A     L 0.0;
      AN    #IN_TRANSFER_BASLADI;
      A(;
      L     3.000000e+00;
      L     #O_SCALE_BASINC_OUT;
      <R;
      );
      A(;
      L     #IN_SET_BASINC;
      L     #O_SCALE_BASINC_OUT;
      >R;
      );
      JNB   _00d;
      L     5.000000e+01;
      T     #ST_OUT_PID_MAN;
_00d: NOP   0;
      A     L 0.0;
      AN    #IN_TRANSFER_BASLADI;
      A(;
      L     #ST_SET_ADD_BASINC_02;
      L     #O_SCALE_BASINC_OUT;
      <=R;
      );
      JNB   _00e;
      L     0.000000e+00;
      T     #ST_OUT_PID_MAN;
_00e: NOP   0;
      A     L 0.0;
      A     #IN_TRANSFER_BASLADI;
      JNB   _00f;
      L     9.000000e+01;
      T     #ST_OUT_PID_MAN;
_00f: NOP   0;
NETWORK
TITLE = Adim 1 - Pisim Süresi
      L     #STATUS;
      L     1;
      ==I;
      =     L 0.0;
      A(;
      A     L 0.0;
      A     #st_basinc_ok_sure_basla;
      L     #IN_PISIM_SURESI;
      T     LD 1;
      TAK;
      T     LD 5;
      L     #IN_TIMER_PISIRME;
      T     LW 9;
      L     LD 5;
      L     LD 1;
      SD    T [LW 9];
      NOP   0;
      NOP   0;
      NOP   0;
      T     LD 1;
      TAK;
      T     LD 5;
      L     #IN_TIMER_PISIRME;
      T     LW 9;
      L     LD 5;
      L     LD 1;
      A     T [LW 9];
      );
      JNB   _010;
      L     2;
      T     #STATUS;
_010: NOP   0;
      A     L 0.0;
      A(;
      O(;
      L     #O_SCALE_BASINC_OUT;
      L     #IN_SET_BASINC;
      >=R;
      );
      O     #st_basinc_ok_sure_basla;
      );
      =     #st_basinc_ok_sure_basla;
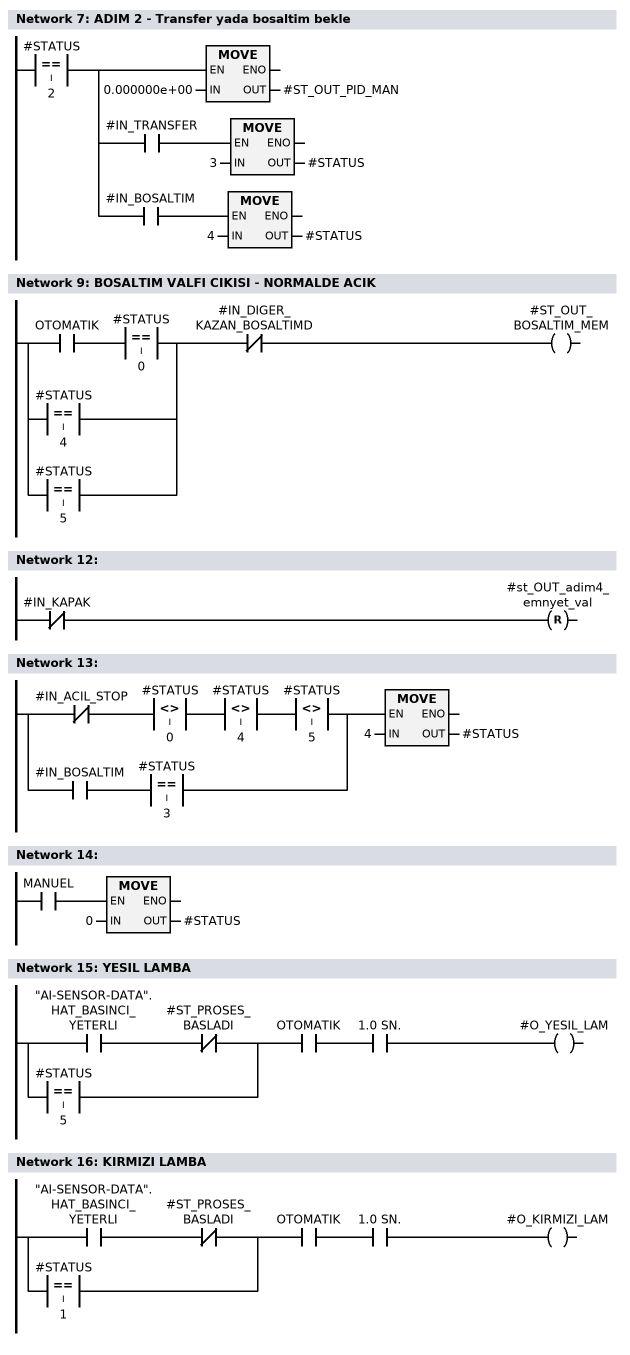
NETWORK
TITLE = ADIM 2 - Transfer yada bosaltim bekle
//1- Adim 2 Transfer ya da bosaltim bekle
//2- Oransal Vanayi kapali tut
      L     #STATUS;
      L     2;
      ==I;
      =     L 0.0;
      A     L 0.0;
      JNB   _011;
      L     0.000000e+00;
      T     #ST_OUT_PID_MAN;
_011: NOP   0;
      A     L 0.0;
      A     #IN_TRANSFER;
      JNB   _012;
      L     3;
      T     #STATUS;
_012: NOP   0;
      A     L 0.0;
      A     #IN_BOSALTIM;
      JNB   _013;
      L     4;
      T     #STATUS;
_013: NOP   0;
NETWORK
TITLE = Adim 3 - Transfer islemi
//1- Diger kazan hazir oldugunda transfer islmeini baslat
      A(;
      L     #STATUS;
      L     3;
      ==I;
      );
      A     #IN_TRANSFERE_HAZIR;
      JNB   _014;
      L     9.000000e+01;
      T     #ST_OUT_PID_MAN;
      SET;
      SAVE;
      CLR;
_014: A     BR;
      =     L 0.0;
      A     L 0.0;
      BLD   102;
      =     #O_TRANSFER_YAPILIYOR;
      A(;
      A     L 0.0;
      L     S5T#23S;
      T     LD 1;
      TAK;
      T     LD 5;
      L     #IN_TIMER_500MS_2;
      T     LW 9;
      L     LD 5;
      L     LD 1;
      SD    T [LW 9];
      NOP   0;
      NOP   0;
      NOP   0;
      T     LD 1;
      TAK;
      T     LD 5;
      L     #IN_TIMER_500MS_2;
      T     LW 9;
      L     LD 5;
      L     LD 1;
      A     T [LW 9];
      );
      JNB   _015;
      L     4;
      T     #STATUS;
_015: NOP   0;
NETWORK
TITLE = BOSALTIM VALFI CIKISI - NORMALDE ACIK
//1- Adim 1,2 ve 3 te bosaltim valfini kapat
//2- Adim 0 ve 4 te bosaltim valfi acik olacak
      A(;
      A     "OTOMATIK";
      A(;
      L     #STATUS;
      L     0;
      ==I;
      );
      O(;
      L     #STATUS;
      L     4;
      ==I;
      );
      O(;
      L     #STATUS;
      L     5;
      ==I;
      );
      );
      AN    #IN_DIGER_KAZAN_BOSALTIMD;
      =     #ST_OUT_BOSALTIM_MEM;
NETWORK
TITLE = Adim 4 - Bosaltim Adimi
      L     #STATUS;
      L     4;
      ==I;
      =     L 0.0;
      A     L 0.0;
      JNB   _016;
      L     0.000000e+00;
      T     #ST_OUT_PID_MAN;
_016: NOP   0;
      A     L 0.0;
      BLD   102;
      =     #ST_KAZAN_BOSALTIMDA;
      A     L 0.0;
      A(;
      L     #O_SCALE_BASINC_OUT;
      L     1.000000e-01;
      <=R;
      );
      =     L 0.1;
      A     L 0.1;
      BLD   102;
      S     #st_OUT_adim4_emnyet_val;
      A(;
      A     L 0.1;
      L     S5T#5S;
      T     LD 1;
      TAK;
      T     LD 5;
      L     #IN_DELAY_BITISI_BEKLE;
      T     LW 9;
      L     LD 5;
      L     LD 1;
      SD    T [LW 9];
      NOP   0;
      NOP   0;
      NOP   0;
      T     LD 1;
      TAK;
      T     LD 5;
      L     #IN_DELAY_BITISI_BEKLE;
      T     LW 9;
      L     LD 5;
      L     LD 1;
      A     T [LW 9];
      );
      JNB   _017;
      L     5;
      T     #STATUS;
_017: NOP   0;
NETWORK
TITLE = KAPAK AÇILMASINI BEKLE
      A(;
      A(;
      L     #STATUS;
      L     5;
      ==I;
      );
      L     S5T#1S;
      T     LD 0;
      TAK;
      T     LD 4;
      L     #IN_DELAY_BIRAZ_BEKLE;
      T     LW 8;
      L     LD 4;
      L     LD 0;
      SD    T [LW 8];
      NOP   0;
      NOP   0;
      NOP   0;
      T     LD 0;
      TAK;
      T     LD 4;
      L     #IN_DELAY_BIRAZ_BEKLE;
      T     LW 8;
      L     LD 4;
      L     LD 0;
      A     T [LW 8];
      );
      AN    #IN_KAPAK;
      JNB   _018;
      L     0;
      T     #STATUS;
_018: NOP   0;
NETWORK
TITLE =
      AN    #IN_KAPAK;
      R     #st_OUT_adim4_emnyet_val;
NETWORK
TITLE =
//1- Acil Stop ile 1,2 ve 3. adimda ise bosaltim adimina git 
//2- 3. adimda bosalt butonu ile bosaltim yapabilsin  
      A(;
      AN    #IN_ACIL_STOP;
      A(;
      L     #STATUS;
      L     0;
      <>I;
      );
      A(;
      L     #STATUS;
      L     4;
      <>I;
      );
      A(;
      L     #STATUS;
      L     5;
      <>I;
      );
      O;
      A     #IN_BOSALTIM;
      A(;
      L     #STATUS;
      L     3;
      ==I;
      );
      );
      JNB   _019;
      L     4;
      T     #STATUS;
_019: NOP   0;
NETWORK
TITLE =
      A     "MANUEL";
      JNB   _01a;
      L     0;
      T     #STATUS;
_01a: NOP   0;
NETWORK
TITLE = YESIL LAMBA
      A(;
      A     "AI-SENSOR-DATA".HAT_BASINCI_YETERLI;
      AN    #ST_PROSES_BASLADI;
      O(;
      L     #STATUS;
      L     5;
      ==I;
      );
      );
      A     "OTOMATIK";
      A     "1.0 SN.";
      =     #O_YESIL_LAM;
NETWORK
TITLE = KIRMIZI LAMBA
      A(;
      A     "AI-SENSOR-DATA".HAT_BASINCI_YETERLI;
      AN    #ST_PROSES_BASLADI;
      O(;
      L     #STATUS;
      L     1;
      ==I;
      );
      );
      A     "OTOMATIK";
      A     "1.0 SN.";
      =     #O_KIRMIZI_LAM;
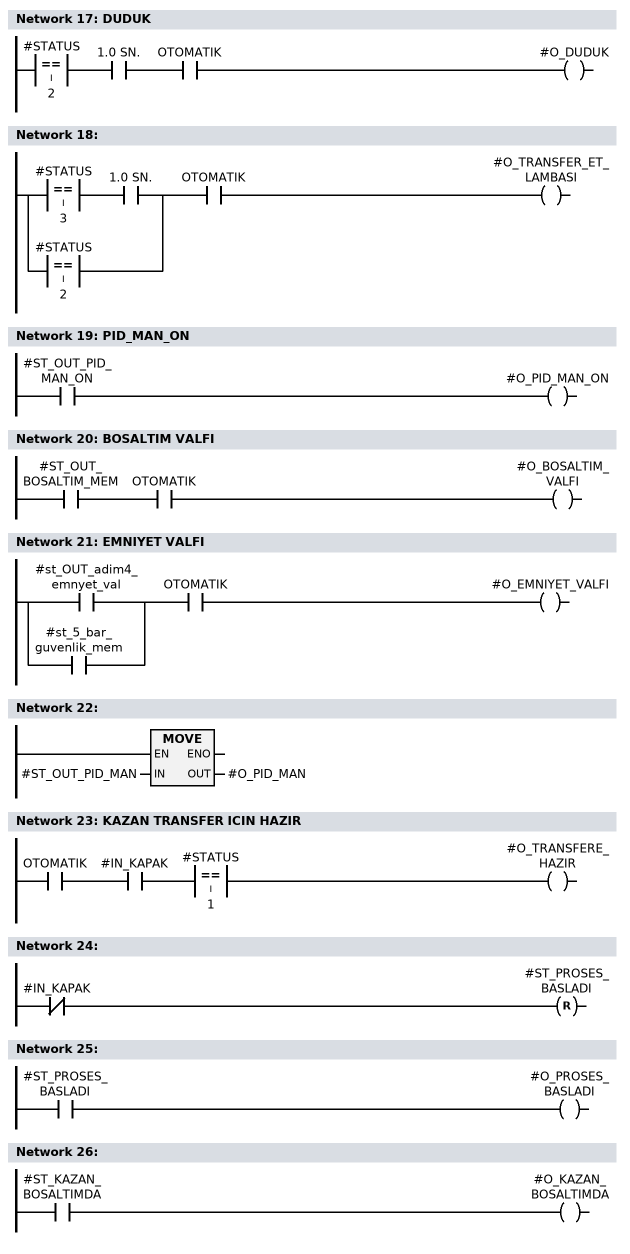
NETWORK
TITLE = DUDUK
      A(;
      L     #STATUS;
      L     2;
      ==I;
      );
      A     "1.0 SN.";
      A     "OTOMATIK";
      =     #O_DUDUK;
NETWORK
TITLE =
      A(;
      A(;
      L     #STATUS;
      L     3;
      ==I;
      );
      A     "1.0 SN.";
      O(;
      L     #STATUS;
      L     2;
      ==I;
      );
      );
      A     "OTOMATIK";
      =     #O_TRANSFER_ET_LAMBASI;
NETWORK
TITLE = PID_MAN_ON 
      A     #ST_OUT_PID_MAN_ON;
      =     #O_PID_MAN_ON;
NETWORK
TITLE = BOSALTIM VALFI
      A     #ST_OUT_BOSALTIM_MEM;
      A     "OTOMATIK";
      =     #O_BOSALTIM_VALFI;
NETWORK
TITLE = EMNIYET VALFI
      A(;
      O     #st_OUT_adim4_emnyet_val;
      O     #st_5_bar_guvenlik_mem;
      );
      A     "OTOMATIK";
      =     #O_EMNIYET_VALFI;
NETWORK
TITLE =
      L     #ST_OUT_PID_MAN;
      T     #O_PID_MAN;
      NOP   0;
NETWORK
TITLE = KAZAN TRANSFER ICIN HAZIR
      A     "OTOMATIK";
      A     #IN_KAPAK;
      A(;
      L     #STATUS;
      L     1;
      ==I;
      );
      =     #O_TRANSFERE_HAZIR;
NETWORK
TITLE =
      AN    #IN_KAPAK;
      R     #ST_PROSES_BASLADI;
NETWORK
TITLE =
      A     #ST_PROSES_BASLADI;
      =     #O_PROSES_BASLADI;
NETWORK
TITLE =
      A     #ST_KAZAN_BOSALTIMDA;
      =     #O_KAZAN_BOSALTIMDA;
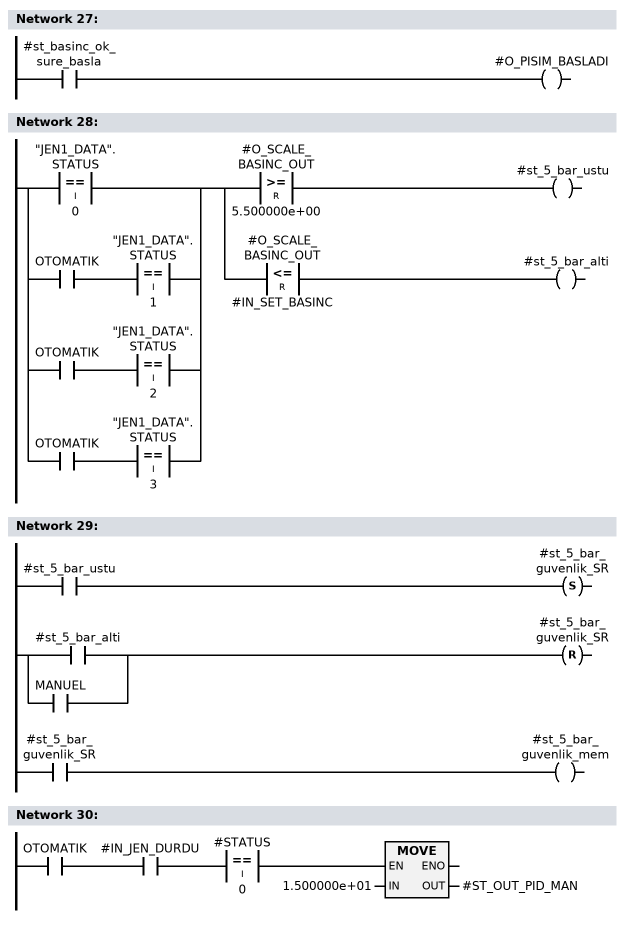
NETWORK
TITLE =
      A     #st_basinc_ok_sure_basla;
      =     #O_PISIM_BASLADI;
NETWORK
TITLE =
//Otoklav 5.5 bar'a geldiginde emniyet vantilini ac ve sete düþtügünde tekrar 
//emniyet ventilini kapat 
      O(;
      L     "JEN1_DATA".STATUS;
      L     0;
      ==I;
      );
      O;
      A     "OTOMATIK";
      A(;
      L     "JEN1_DATA".STATUS;
      L     1;
      ==I;
      );
      O;
      A     "OTOMATIK";
      A(;
      L     "JEN1_DATA".STATUS;
      L     2;
      ==I;
      );
      O;
      A     "OTOMATIK";
      A(;
      L     "JEN1_DATA".STATUS;
      L     3;
      ==I;
      );
      =     L 0.0;
      A     L 0.0;
      A(;
      L     #O_SCALE_BASINC_OUT;
      L     5.500000e+00;
      >=R;
      );
      =     #st_5_bar_ustu;
      A     L 0.0;
      A(;
      L     #O_SCALE_BASINC_OUT;
      L     #IN_SET_BASINC;
      <=R;
      );
      =     #st_5_bar_alti;
NETWORK
TITLE =
      A     #st_5_bar_ustu;
      S     #st_5_bar_guvenlik_SR;
      A(;
      O     #st_5_bar_alti;
      O     "MANUEL";
      );
      R     #st_5_bar_guvenlik_SR;
      A     #st_5_bar_guvenlik_SR;
      =     #st_5_bar_guvenlik_mem;
NETWORK
TITLE =
//JENERATORLER DURDUGUNDA BELIRLI SANIYE ORANSAL VANAYI AC HATTA BULUNAN BUHAR 
//TASFIYE EDILSIN
      A     "OTOMATIK";
      A     #IN_JEN_DURDU;
      A(;
      L     #STATUS;
      L     0;
      ==I;
      );
      JNB   _01b;
      L     1.500000e+01;
      T     #ST_OUT_PID_MAN;
_01b: NOP   0;
END_FUNCTION_BLOCK

// FB 41: know-how protected block, not included

FUNCTION_BLOCK "KAZAN_1_PID_KONTROL"	// FB 47
//KAZAN 1 PID BLOGU
VERSION : 0.1
BEGIN
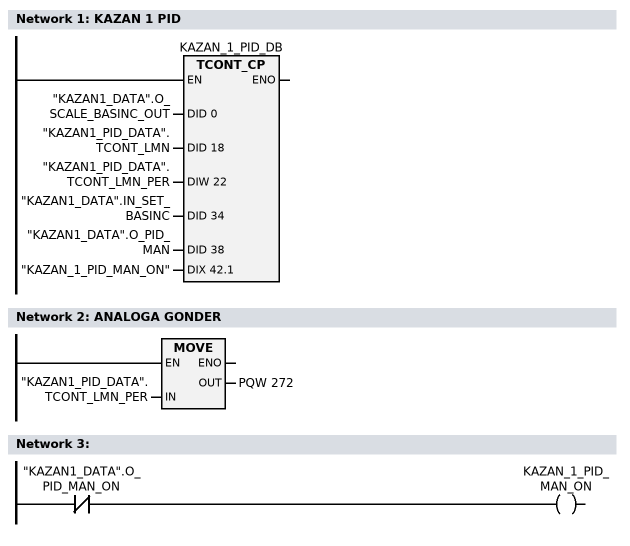
NETWORK
TITLE = KAZAN 1 PID
      CALL  "TCONT_CP" , "KAZAN_1_PID_DB" (
           DID 0                    := "KAZAN1_DATA".O_SCALE_BASINC_OUT,
           DID 18                   := "KAZAN1_PID_DATA".TCONT_LMN,
           DIW 22                   := "KAZAN1_PID_DATA".TCONT_LMN_PER,
           DID 34                   := "KAZAN1_DATA".IN_SET_BASINC,
           DID 38                   := "KAZAN1_DATA".O_PID_MAN,
           DIX 42.1                 := "KAZAN_1_PID_MAN_ON");
      NOP   0;
NETWORK
TITLE = ANALOGA GONDER
      L     "KAZAN1_PID_DATA".TCONT_LMN_PER;
      T     PQW 272;
      NOP   0;
NETWORK
TITLE =
      AN    "KAZAN1_DATA".O_PID_MAN_ON;
      =     "KAZAN_1_PID_MAN_ON";
NETWORK
TITLE =
END_FUNCTION_BLOCK

FUNCTION_BLOCK "KAZAN_2_PID_KONTROL"	// FB 48
VERSION : 0.1
BEGIN
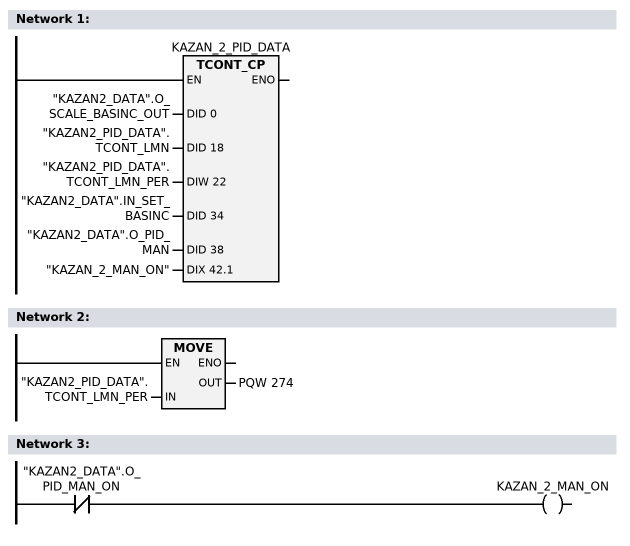
NETWORK
TITLE =
      CALL  "TCONT_CP" , "KAZAN_2_PID_DATA" (
           DID 0                    := "KAZAN2_DATA".O_SCALE_BASINC_OUT,
           DID 18                   := "KAZAN2_PID_DATA".TCONT_LMN,
           DIW 22                   := "KAZAN2_PID_DATA".TCONT_LMN_PER,
           DID 34                   := "KAZAN2_DATA".IN_SET_BASINC,
           DID 38                   := "KAZAN2_DATA".O_PID_MAN,
           DIX 42.1                 := "KAZAN_2_MAN_ON");
      NOP   0;
NETWORK
TITLE =
      L     "KAZAN2_PID_DATA".TCONT_LMN_PER;
      T     PQW 274;
      NOP   0;
NETWORK
TITLE =
      AN    "KAZAN2_DATA".O_PID_MAN_ON;
      =     "KAZAN_2_MAN_ON";
END_FUNCTION_BLOCK

FUNCTION_BLOCK "JEN1_PID_KONTROL"	// FB 49
//GAIN: 8.21488
//TI : 2.11452
//TD : 0.585774
//DERIVATIVE FACTOR: 5
//UPPER LIMIT : 80
//FACTOR : -1
//OFFSET : 100
VERSION : 0.1
VAR
  TCONT_C_MAN : REAL ;
  TCONT_C_MAN_ON : BOOL ;
  TCONT_C_LMN : REAL ;
  TCONT_C_LMN_PER : INT ;
END_VAR
BEGIN
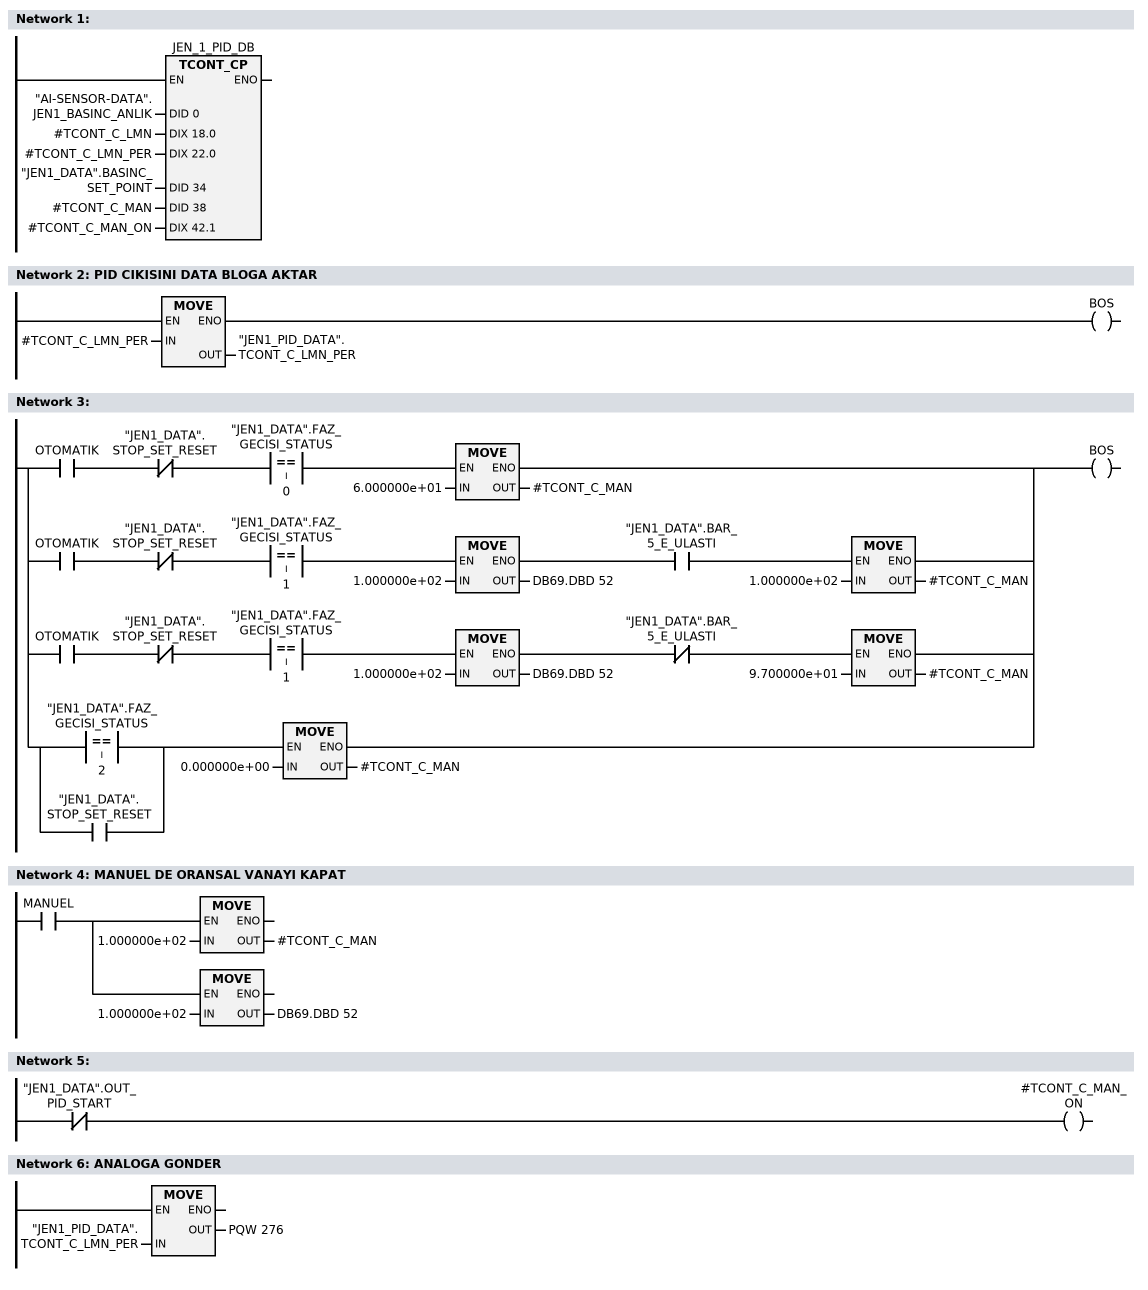
NETWORK
TITLE =
      CALL  "TCONT_CP" , "JEN_1_PID_DB" (
           DID 0                    := "AI-SENSOR-DATA".JEN1_BASINC_ANLIK,
           DIX 18.0                 := #TCONT_C_LMN,
           DIX 22.0                 := #TCONT_C_LMN_PER,
           DID 34                   := "JEN1_DATA".BASINC_SET_POINT,
           DID 38                   := #TCONT_C_MAN,
           DIX 42.1                 := #TCONT_C_MAN_ON);
      NOP   0;
NETWORK
TITLE = PID CIKISINI DATA BLOGA AKTAR
//SICAKLIK_2_OK  KISMINDAN PQW278 SILINDI. YERINE DB20.DBD0 BASINC SET DEGERI
//EKLENDI
      L     #TCONT_C_LMN_PER;
      T     "JEN1_PID_DATA".TCONT_C_LMN_PER;
      SET;
      SAVE;
      CLR;
      A     BR;
      =     "BOS";
NETWORK
TITLE =
//FAZ DURUMUNA GORE MAN DEGERINI AYARLA
//FAZ 1 - MAN CIKIS OLARAK 40 GONDER- 40 TAN BASLAMASI ICIN
//FAZ 2 - TAMAMEN KAPANMASI ICIN 0 GONDER (PID MAUELDE)
//FAZ 3 - GUVENLIK SORUNLARINDA VANAYI TAMAMEN AC
      O(;
      A     "OTOMATIK";
      AN    "JEN1_DATA".STOP_SET_RESET;
      A(;
      L     "JEN1_DATA".FAZ_GECISI_STATUS;
      L     0;
      ==I;
      );
      JNB   _001;
      L     6.000000e+01;
      T     #TCONT_C_MAN;
      SET;
      SAVE;
      CLR;
_001: A     BR;
      );
      O(;
      A(;
      A     "OTOMATIK";
      AN    "JEN1_DATA".STOP_SET_RESET;
      A(;
      L     "JEN1_DATA".FAZ_GECISI_STATUS;
      L     1;
      ==I;
      );
      JNB   _002;
      L     1.000000e+02;
      T     DB69.DBD 52;
      SET;
      SAVE;
      CLR;
_002: A     BR;
      );
      A     "JEN1_DATA".BAR_5_E_ULASTI;
      JNB   _003;
      L     1.000000e+02;
      T     #TCONT_C_MAN;
      SET;
      SAVE;
      CLR;
_003: A     BR;
      );
      O(;
      A(;
      A     "OTOMATIK";
      AN    "JEN1_DATA".STOP_SET_RESET;
      A(;
      L     "JEN1_DATA".FAZ_GECISI_STATUS;
      L     1;
      ==I;
      );
      JNB   _004;
      L     1.000000e+02;
      T     DB69.DBD 52;
      SET;
      SAVE;
      CLR;
_004: A     BR;
      );
      AN    "JEN1_DATA".BAR_5_E_ULASTI;
      JNB   _005;
      L     9.700000e+01;
      T     #TCONT_C_MAN;
      SET;
      SAVE;
      CLR;
_005: A     BR;
      );
      O(;
      A(;
      O(;
      L     "JEN1_DATA".FAZ_GECISI_STATUS;
      L     2;
      ==I;
      );
      O     "JEN1_DATA".STOP_SET_RESET;
      );
      JNB   _006;
      L     0.000000e+00;
      T     #TCONT_C_MAN;
      SET;
      SAVE;
      CLR;
_006: A     BR;
      );
      =     "BOS";
NETWORK
TITLE = MANUEL DE ORANSAL VANAYI KAPAT
      A     "MANUEL";
      =     L 0.0;
      A     L 0.0;
      JNB   _007;
      L     1.000000e+02;
      T     #TCONT_C_MAN;
_007: NOP   0;
      A     L 0.0;
      JNB   _008;
      L     1.000000e+02;
      T     DB69.DBD 52;
_008: NOP   0;
NETWORK
TITLE =
      AN    "JEN1_DATA".OUT_PID_START;
      =     #TCONT_C_MAN_ON;
NETWORK
TITLE = ANALOGA GONDER
      L     "JEN1_PID_DATA".TCONT_C_LMN_PER;
      T     PQW 276;
      NOP   0;
END_FUNCTION_BLOCK

FUNCTION_BLOCK "JEN2_PID_KONTROL"	// FB 50
//GAIN: 8.21488
//TI : 2.11452
//TD : 0.585774
//DERIVATIVE FACTOR: 5
//UPPER LIMIT : 80
//FACTOR : -1
//OFFSET : 100
VERSION : 0.1
VAR
  TCONT_C_LMN : REAL ;
  TCONT_C_LMN_PER : INT ;
  TCONT_C_MAN : REAL ;
  TCONT_C_MAN_ON : BOOL ;
  Ris_5_Bar : BOOL ;
END_VAR
BEGIN
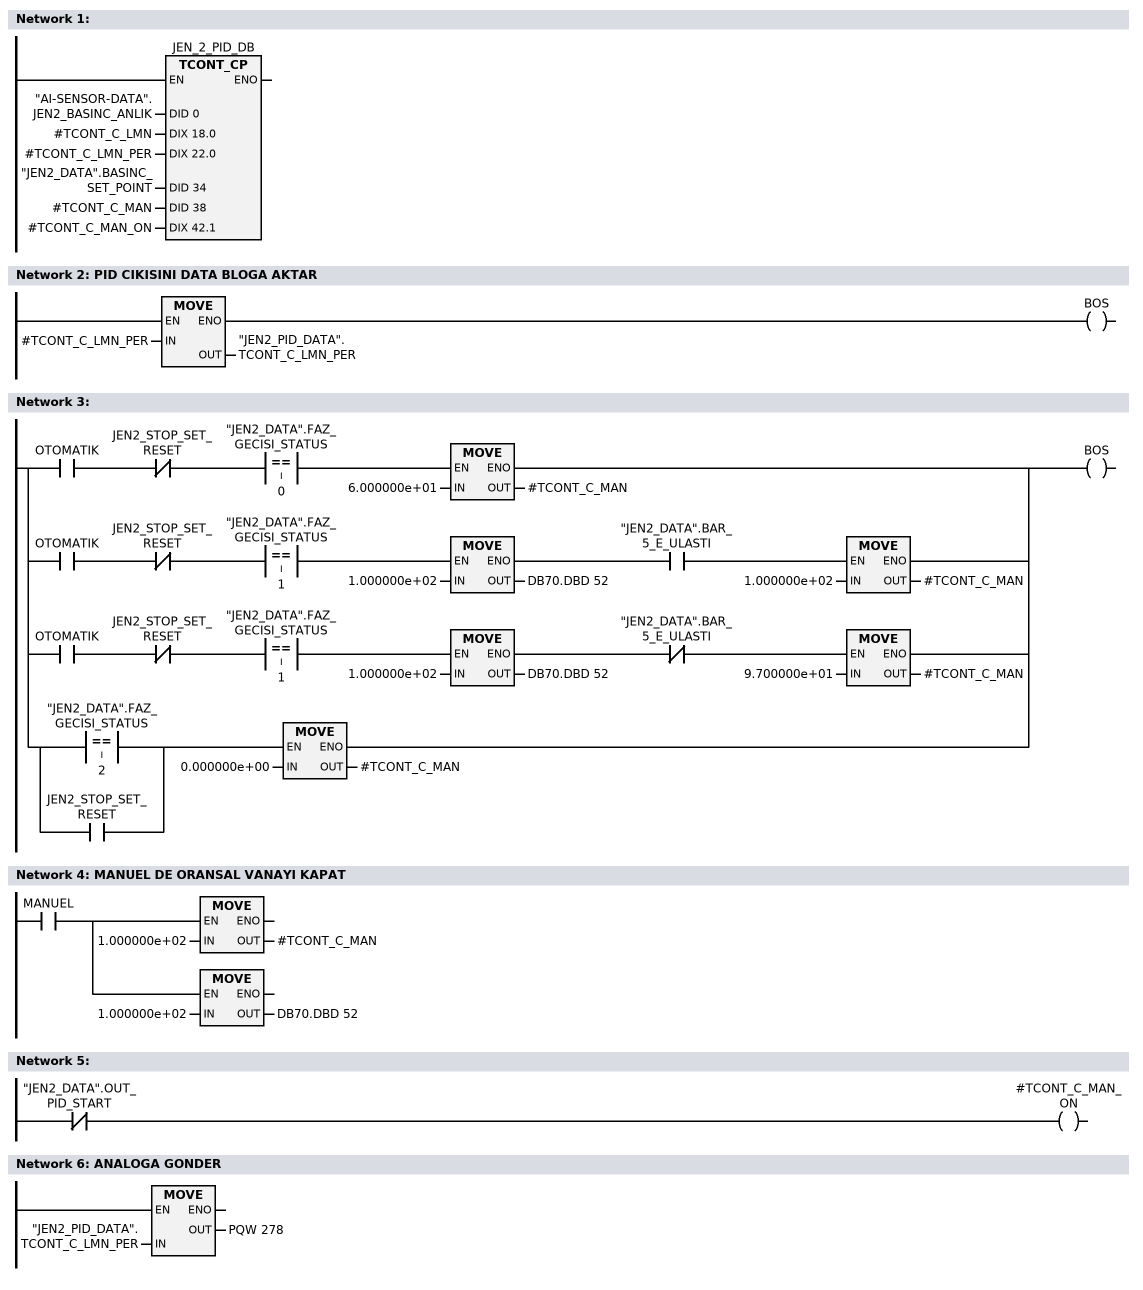
NETWORK
TITLE =
      CALL  "TCONT_CP" , "JEN_2_PID_DB" (
           DID 0                    := "AI-SENSOR-DATA".JEN2_BASINC_ANLIK,
           DIX 18.0                 := #TCONT_C_LMN,
           DIX 22.0                 := #TCONT_C_LMN_PER,
           DID 34                   := "JEN2_DATA".BASINC_SET_POINT,
           DID 38                   := #TCONT_C_MAN,
           DIX 42.1                 := #TCONT_C_MAN_ON);
      NOP   0;
NETWORK
TITLE = PID CIKISINI DATA BLOGA AKTAR
//SICAKLIK_2_OK  KISMINDAN PQW278 SILINDI. YERINE DB20.DBD0 BASINC SET DEGERI
//EKLENDI
      L     #TCONT_C_LMN_PER;
      T     "JEN2_PID_DATA".TCONT_C_LMN_PER;
      SET;
      SAVE;
      CLR;
      A     BR;
      =     "BOS";
NETWORK
TITLE =
//FAZ DURUMUNA GORE MAN DEGERINI AYARLA
//FAZ 1 - MAN CIKIS OLARAK 40 GONDER- 40 TAN BASLAMASI ICIN
//FAZ 2 - TAMAMEN KAPANMASI ICIN 0 GONDER (PID MAUELDE)
//FAZ 3 - GUVENLIK SORUNLARINDA VANAYI TAMAMEN AC
      O(;
      A     "OTOMATIK";
      AN    "JEN2_STOP_SET_RESET";
      A(;
      L     "JEN2_DATA".FAZ_GECISI_STATUS;
      L     0;
      ==I;
      );
      JNB   _001;
      L     6.000000e+01;
      T     #TCONT_C_MAN;
      SET;
      SAVE;
      CLR;
_001: A     BR;
      );
      O(;
      A(;
      A     "OTOMATIK";
      AN    "JEN2_STOP_SET_RESET";
      A(;
      L     "JEN2_DATA".FAZ_GECISI_STATUS;
      L     1;
      ==I;
      );
      JNB   _002;
      L     1.000000e+02;
      T     DB70.DBD 52;
      SET;
      SAVE;
      CLR;
_002: A     BR;
      );
      A     "JEN2_DATA".BAR_5_E_ULASTI;
      JNB   _003;
      L     1.000000e+02;
      T     #TCONT_C_MAN;
      SET;
      SAVE;
      CLR;
_003: A     BR;
      );
      O(;
      A(;
      A     "OTOMATIK";
      AN    "JEN2_STOP_SET_RESET";
      A(;
      L     "JEN2_DATA".FAZ_GECISI_STATUS;
      L     1;
      ==I;
      );
      JNB   _004;
      L     1.000000e+02;
      T     DB70.DBD 52;
      SET;
      SAVE;
      CLR;
_004: A     BR;
      );
      AN    "JEN2_DATA".BAR_5_E_ULASTI;
      JNB   _005;
      L     9.700000e+01;
      T     #TCONT_C_MAN;
      SET;
      SAVE;
      CLR;
_005: A     BR;
      );
      O(;
      A(;
      O(;
      L     "JEN2_DATA".FAZ_GECISI_STATUS;
      L     2;
      ==I;
      );
      O     "JEN2_STOP_SET_RESET";
      );
      JNB   _006;
      L     0.000000e+00;
      T     #TCONT_C_MAN;
      SET;
      SAVE;
      CLR;
_006: A     BR;
      );
      =     "BOS";
NETWORK
TITLE = MANUEL DE ORANSAL VANAYI KAPAT
      A     "MANUEL";
      =     L 0.0;
      A     L 0.0;
      JNB   _007;
      L     1.000000e+02;
      T     #TCONT_C_MAN;
_007: NOP   0;
      A     L 0.0;
      JNB   _008;
      L     1.000000e+02;
      T     DB70.DBD 52;
_008: NOP   0;
NETWORK
TITLE =
      AN    "JEN2_DATA".OUT_PID_START;
      =     #TCONT_C_MAN_ON;
NETWORK
TITLE = ANALOGA GONDER
      L     "JEN2_PID_DATA".TCONT_C_LMN_PER;
      T     PQW 278;
      NOP   0;
END_FUNCTION_BLOCK

// FB 58: know-how protected block, not included

FUNCTION_BLOCK "KAZAN_1_KONTROL"	// FB 94
VERSION : 0.1
BEGIN
NETWORK
TITLE =
      CALL  "KAZAN_ORTAK" , DB 120 (
           IN_ACIL_STOP             := "KAZAN1_ACIL_STOP",
           IN_START                 := "KAZAN1_START",
           IN_TRANSFER              := "KAZAN1_TRANSFER",
           IN_BOSALTIM              := "KAZAN1_BOSALTIM",
           IN_KAPAK                 := "KAZAN1_KAPAK_SW",
           IN_JENS_OK               := "KAZAN1_DATA".IN_JEN_OK,
           IN_TRANSFERE_HAZIR       := "KAZAN1_DATA".IN_DIGER_KAZ_TRANS_HAZIR,
           IN_PISIM_SURESI          := "KAZAN1_DATA".IN_PISIM_SURESI,
           IN_SCALE_BASINC_PER      := "KAZAN1_DATA".IN_SCALE_BASINC_PER,
           IN_SET_BASINC            := "KAZAN1_DATA".IN_SET_BASINC,
           IN_DIGER_KAZAN_BASINCI   := "KAZAN1_DATA".IN_DIGER_KAZAN_BASINCI,
           IN_TIMER_500MS           := "500ms_delay1",
           IN_TIMER_1S              := "1s Delay",
           IN_TIMER_PISIRME         := "Pisim_Suresi",
           IN_TIMER_500MS_2         := "500ms_delay",
           IN_TIMER_7S              := "s_offt_7s_delay",
           IN_SCALE_HI_LIM          := 1.000000e+01,
           IN_SCALE_LO_LIM          := 0.000000e+00,
           IN_SCALE_SICAKLIK_HI_LIM := 2.000000e+02,
           IN_SCALE_SICAKLIK_LO_LIM := 0.000000e+00,
           IN_SCALE_SICAKLIK_PER    := "KAZAN1_DATA".IN_SCALE_SICAKLIK_PER,
           IN_DIGER_KAZAN_BOSALTIMD := "KAZAN1_DATA".IN_DIGER_KAZ_BOSALTIMDA,
           IN_TRANSFER_BASLADI      := "KAZAN1_DATA".IN_DIGER_KAZ_TRANSFERDE,
           IN_JEN_DURDU             := "ORTAK_DATA".OTO_ISLEM_BITTI_VANA_AC,
           IN_DELAY_BITISI_BEKLE    := "OTO_1_DELAY_PISIM_BITTI",
           IN_DELAY_BIRAZ_BEKLE     := "DELAY_ADIM5_BEKLE",
           O_YESIL_LAM              := "KAZAN1_YESIL_LAMBA",
           O_KIRMIZI_LAM            := "KAZAN1_KIRMIZI_LAMBA",
           O_DUDUK                  := "KAZAN1_DUDUK",
           O_BOSALTIM_VALFI         := "KAZAN1_BOSALTIM_VALFI",
           O_PID_MAN_ON             := "KAZAN1_DATA".O_PID_MAN_ON,
           O_PID_MAN                := "KAZAN1_DATA".O_PID_MAN,
           O_TRANSFER_YAPILIYOR     := "KAZAN1_DATA".O_TRANSFER_YAPILIYOR,
           O_SCALE_BASINC_RET_VAL   := "KAZAN1_DATA".O_SCALE_BASINC_RET_VAL,
           O_SCALE_BASINC_OUT       := "KAZAN1_DATA".O_SCALE_BASINC_OUT,
           O_EMNIYET_VALFI          := "KAZAN1_EMN_VALFI_BOS",
           O_TRANSFERE_HAZIR        := "KAZAN1_DATA".O_TRANSFERE_HAZIR,
           O_SCALE_SICAKLIK_RET_VAL := "KAZAN1_DATA".O_SCALE_SICAKLIK_RET_VAL,
           O_SCALE_SICAKLIK_OUT     := "KAZAN1_DATA".O_SCALE_SICAKLIK_OUT,
           O_TRANSFER_ET_LAMBASI    := "KAZAN1_TRANS_BUT_LAMBASI",
           O_PROSES_BASLADI         := M 300.0,
           O_KAZAN_BOSALTIMDA       := "KAZAN1_DATA".O_KAZAN_BOSALTIMDA,
           O_PISIM_BASLADI          := "KAZAN1_DATA".O_PISIM_BASLADI,
           STATUS                   := "KAZAN1_DATA".IN_STATUS);
//       O_YESIL_LAM             :="KAZAN1_YESIL_LAMBA"
//       O_KIRMIZI_LAM           :="KAZAN1_KIRMIZI_LAMBA"
//       O_DUDUK                 :="KAZAN1_DUDUK"
//       O_BOSALTIM_VALFI        :="KAZAN1_BOSALTIM_VALFI"
//       O_PID_MAN_ON            :="KAZAN1_DATA".O_PID_MAN_ON
//       O_PID_MAN               :="KAZAN1_DATA".O_PID_MAN
//       O_TRANSFER_YAPILIYOR    :="KAZAN1_DATA".O_TRANSFER_YAPILIYOR
//       O_SCALE_BASINC_RET_VAL  :="KAZAN1_DATA".O_SCALE_BASINC_RET_VAL
//       O_SCALE_BASINC_OUT      :="KAZAN1_DATA".O_SCALE_BASINC_OUT
//       O_EMNIYET_VALFI         :="KAZAN1_EMN_VALFI_BOS"
//       O_TRANSFERE_HAZIR       :="KAZAN1_DATA".O_TRANSFERE_HAZIR
//       O_SCALE_SICAKLIK_RET_VAL:="KAZAN1_DATA".O_SCALE_SICAKLIK_RET_VAL
//       O_SCALE_SICAKLIK_OUT    :="KAZAN1_DATA".O_SCALE_SICAKLIK_OUT
//       O_TRANSFER_ET_LAMBASI   :="KAZAN1_TRANS_BUT_LAMBASI"
//       O_PROSES_BASLADI        :=M300.0
//       O_KAZAN_BOSALTIMDA      :="KAZAN1_DATA".O_KAZAN_BOSALTIMDA
//       O_PISIM_BASLADI         :="KAZAN1_DATA".O_PISIM_BASLADI
//       STATUS                  :="KAZAN1_DATA".IN_STATUS
NETWORK
TITLE = GIRIS-CIKIS
      A     "KAZAN2_DATA".O_TRANSFERE_HAZIR;
      =     "KAZAN1_DATA".IN_DIGER_KAZ_TRANS_HAZIR;
      L     PIW 272;
      T     "KAZAN1_DATA".IN_SCALE_BASINC_PER;
      L     PIW 274;
      T     "KAZAN1_DATA".IN_SCALE_SICAKLIK_PER;
      L     "KAZAN2_DATA".O_SCALE_BASINC_OUT;
      T     "KAZAN1_DATA".IN_DIGER_KAZAN_BASINCI;
      O     "JEN1_DATA".JEN1_HAZIR;
      O     "JEN2_DATA".JEN2_HAZIR;
      =     "KAZAN1_DATA".IN_JEN_OK;
      A     "KAZAN2_DATA".O_KAZAN_BOSALTIMDA;
      =     "KAZAN1_DATA".IN_DIGER_KAZ_BOSALTIMDA;
      A     "KAZAN2_DATA".O_TRANSFER_YAPILIYOR;
      =     "KAZAN1_DATA".IN_DIGER_KAZ_TRANSFERDE;
END_FUNCTION_BLOCK

FUNCTION_BLOCK "KAZAN_2_KONTROL"	// FB 95
VERSION : 0.1
BEGIN
NETWORK
TITLE =
      CALL  "KAZAN_ORTAK" , DB 230 (
           IN_ACIL_STOP             := "KAZAN2_ACIL_STOP",
           IN_START                 := "KAZAN2_START",
           IN_TRANSFER              := "KAZAN2_TRANSFER",
           IN_BOSALTIM              := "KAZAN2_BOSALTIM",
           IN_KAPAK                 := "KAZAN2_KAPAK_SW",
           IN_JENS_OK               := "KAZAN2_DATA".IN_JEN_OK,
           IN_TRANSFERE_HAZIR       := "KAZAN2_DATA".IN_DIGER_KAZ_TRANS_HAZIR,
           IN_PISIM_SURESI          := "KAZAN2_DATA".IN_PISIM_SURESI,
           IN_SCALE_BASINC_PER      := "KAZAN2_DATA".IN_SCALE_BASINC_PER,
           IN_SET_BASINC            := "KAZAN2_DATA".IN_SET_BASINC,
           IN_DIGER_KAZAN_BASINCI   := "KAZAN2_DATA".IN_DIGER_KAZAN_BASINCI,
           IN_TIMER_500MS           := "500ms_delay_kazan_2",
           IN_TIMER_1S              := "1ms_delay_kazan_2",
           IN_TIMER_PISIRME         := "kazan_2_pisirme_delay",
           IN_TIMER_500MS_2         := "kazan_2_500ms_delay",
           IN_TIMER_7S              := "kazan_2_7s_delay",
           IN_SCALE_HI_LIM          := 1.000000e+01,
           IN_SCALE_LO_LIM          := 0.000000e+00,
           IN_SCALE_SICAKLIK_HI_LIM := 2.000000e+02,
           IN_SCALE_SICAKLIK_LO_LIM := 0.000000e+00,
           IN_SCALE_SICAKLIK_PER    := "KAZAN2_DATA".IN_SCALE_SICAKLIK_PER,
           IN_DIGER_KAZAN_BOSALTIMD := "KAZAN2_DATA".IN_DIGER_KAZ_BOSALTIMDA,
           IN_TRANSFER_BASLADI      := "KAZAN2_DATA".IN_DIGER_KAZ_TRANSFERDE,
           IN_JEN_DURDU             := "ORTAK_DATA".OTO_ISLEM_BITTI_VANA_AC,
           IN_DELAY_BITISI_BEKLE    := "OTO_2_DELAY_BITIS",
           IN_DELAY_BIRAZ_BEKLE     := "DELAY_ADIM5_BEKLE2",
           O_YESIL_LAM              := "KAZAN2_YESIL_LAMBA",
           O_KIRMIZI_LAM            := "KAZAN2_KIRMIZI_LAMBA",
           O_DUDUK                  := "KAZAN2_DUDUK",
           O_BOSALTIM_VALFI         := "KAZAN2_BOSALTIM_VALFI",
           O_PID_MAN_ON             := "KAZAN2_DATA".O_PID_MAN_ON,
           O_PID_MAN                := "KAZAN2_DATA".O_PID_MAN,
           O_TRANSFER_YAPILIYOR     := "KAZAN2_DATA".O_TRANSFER_YAPILIYOR,
           O_SCALE_BASINC_RET_VAL   := "KAZAN2_DATA".O_SCALE_BASINC_RET_VAL,
           O_SCALE_BASINC_OUT       := "KAZAN2_DATA".O_SCALE_BASINC_OUT,
           O_EMNIYET_VALFI          := "KAZAN2_EMN_VALFI_BOS",
           O_TRANSFERE_HAZIR        := "KAZAN2_DATA".O_TRANSFERE_HAZIR,
           O_SCALE_SICAKLIK_RET_VAL := "KAZAN2_DATA".O_SCALE_SICAKLIK_RET_VAL,
           O_SCALE_SICAKLIK_OUT     := "KAZAN2_DATA".O_SCALE_SICAKLIK_OUT,
           O_TRANSFER_ET_LAMBASI    := "KAZAN2_TRANS_BUT_LAMBASI",
           O_PROSES_BASLADI         := M 300.1,
           O_KAZAN_BOSALTIMDA       := "KAZAN2_DATA".O_KAZAN_BOSALTIMDA,
           O_PISIM_BASLADI          := "KAZAN2_DATA".O_PISIM_BASLADI,
           STATUS                   := "KAZAN2_DATA".IN_STATUS);
//       O_YESIL_LAM             :="KAZAN2_YESIL_LAMBA"
//       O_KIRMIZI_LAM           :="KAZAN2_KIRMIZI_LAMBA"
//       O_DUDUK                 :="KAZAN2_DUDUK"
//       O_BOSALTIM_VALFI        :="KAZAN2_BOSALTIM_VALFI"
//       O_PID_MAN_ON            :="KAZAN2_DATA".O_PID_MAN_ON
//       O_PID_MAN               :="KAZAN2_DATA".O_PID_MAN
//       O_TRANSFER_YAPILIYOR    :="KAZAN2_DATA".O_TRANSFER_YAPILIYOR
//       O_SCALE_BASINC_RET_VAL  :="KAZAN2_DATA".O_SCALE_BASINC_RET_VAL
//       O_SCALE_BASINC_OUT      :="KAZAN2_DATA".O_SCALE_BASINC_OUT
//       O_EMNIYET_VALFI         :="KAZAN2_EMN_VALFI_BOS"
//       O_TRANSFERE_HAZIR       :="KAZAN2_DATA".O_TRANSFERE_HAZIR
//       O_SCALE_SICAKLIK_RET_VAL:="KAZAN2_DATA".O_SCALE_SICAKLIK_RET_VAL
//       O_SCALE_SICAKLIK_OUT    :="KAZAN2_DATA".O_SCALE_SICAKLIK_OUT
//       O_TRANSFER_ET_LAMBASI   :="KAZAN2_TRANS_BUT_LAMBASI"
//       O_PROSES_BASLADI        :=M300.1
//       O_KAZAN_BOSALTIMDA      :="KAZAN2_DATA".O_KAZAN_BOSALTIMDA
//       O_PISIM_BASLADI         :="KAZAN2_DATA".O_PISIM_BASLADI
//       STATUS                  :="KAZAN2_DATA".IN_STATUS
NETWORK
TITLE =
      A     "KAZAN1_DATA".O_TRANSFERE_HAZIR;
      =     "KAZAN2_DATA".IN_DIGER_KAZ_TRANS_HAZIR;
      L     PIW 276;
      T     "KAZAN2_DATA".IN_SCALE_BASINC_PER;
      L     PIW 278;
      T     "KAZAN2_DATA".IN_SCALE_SICAKLIK_PER;
      L     "KAZAN1_DATA".O_SCALE_BASINC_OUT;
      T     "KAZAN2_DATA".IN_DIGER_KAZAN_BASINCI;
      O     "JEN1_DATA".JEN1_HAZIR;
      O     "JEN2_DATA".JEN2_HAZIR;
      =     "KAZAN2_DATA".IN_JEN_OK;
      A     "KAZAN1_DATA".O_KAZAN_BOSALTIMDA;
      =     "KAZAN2_DATA".IN_DIGER_KAZ_BOSALTIMDA;
      A     "KAZAN1_DATA".O_TRANSFER_YAPILIYOR;
      =     "KAZAN2_DATA".IN_DIGER_KAZ_TRANSFERDE;
END_FUNCTION_BLOCK

FUNCTION_BLOCK "JEN1_KONTROL_BLOGU"	// FB 98
VERSION : 0.1
VAR
  st_Set_100_Derece : BOOL ;
  Set1_OK : BOOL ;
  st_Stop_Trigger : BOOL ;
  st_Stop_Set_Mem : BOOL ;
  st_Sicaklik_Dustu : BOOL ;
END_VAR
VAR_TEMP
  t_Ris_Set_100 : BOOL ;
  t_Ris_Start : BOOL ;
  t_Ris_Status : BOOL ;
  t_Ris_Status2 : BOOL ;
  t_Ris_Status3 : BOOL ;
  t_Ris_Set1_ok : BOOL ;
  t_Ris_Set1_ok_1 : BOOL ;
  t_Ris_Set1_ok_2 : BOOL ;
  t_Ris_Stop : BOOL ;
  t_Ris_Sogutma : BOOL ;
  t_Fall_Sogutma : BOOL ;
  t_Ris_Sicaklik_Dustu : BOOL ;
END_VAR
BEGIN
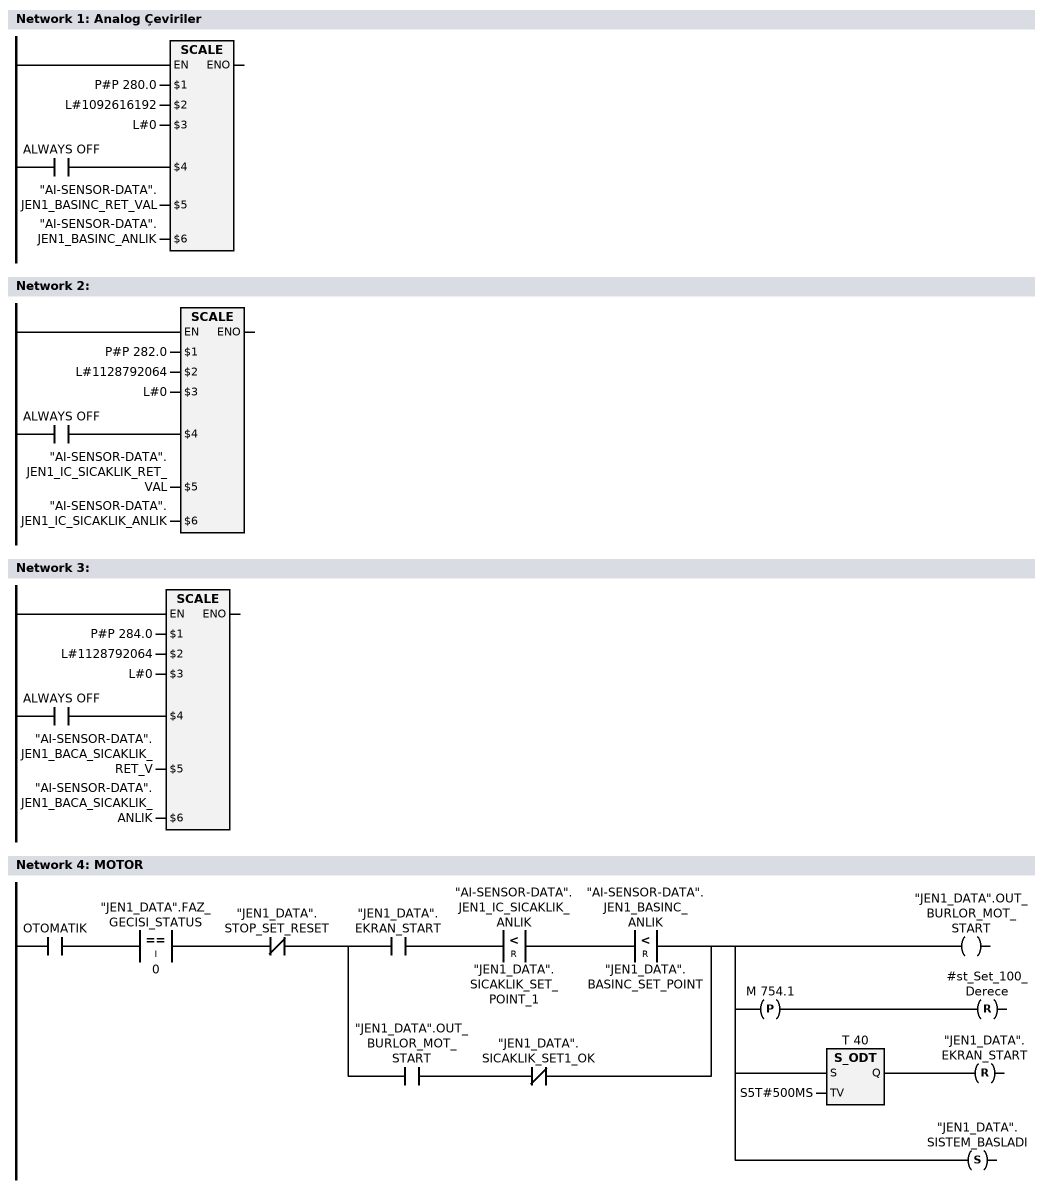
NETWORK
TITLE = Analog Çeviriler
      A     "ALWAYS OFF";
      =     L 2.0;
      BLD   103;
      CALL  "SCALE" (
           $1                       := P#P 280.0,
           $2                       := L#1092616192,
           $3                       := L#0,
           $4                       := L 2.0,
           $5                       := "AI-SENSOR-DATA".JEN1_BASINC_RET_VAL,
           $6                       := "AI-SENSOR-DATA".JEN1_BASINC_ANLIK);
      NOP   0;
NETWORK
TITLE =
      A     "ALWAYS OFF";
      =     L 2.0;
      BLD   103;
      CALL  "SCALE" (
           $1                       := P#P 282.0,
           $2                       := L#1128792064,
           $3                       := L#0,
           $4                       := L 2.0,
           $5                       := "AI-SENSOR-DATA".JEN1_IC_SICAKLIK_RET_VAL,
           $6                       := "AI-SENSOR-DATA".JEN1_IC_SICAKLIK_ANLIK);
      NOP   0;
NETWORK
TITLE =
      A     "ALWAYS OFF";
      =     L 2.0;
      BLD   103;
      CALL  "SCALE" (
           $1                       := P#P 284.0,
           $2                       := L#1128792064,
           $3                       := L#0,
           $4                       := L 2.0,
           $5                       := "AI-SENSOR-DATA".JEN1_BACA_SICAKLIK_RET_V,
           $6                       := "AI-SENSOR-DATA".JEN1_BACA_SICAKLIK_ANLIK);
      NOP   0;
NETWORK
TITLE = MOTOR
      A     "OTOMATIK";
      A(;
      L     "JEN1_DATA".FAZ_GECISI_STATUS;
      L     0;
      ==I;
      );
      AN    "JEN1_DATA".STOP_SET_RESET;
      A(;
      A     "JEN1_DATA".EKRAN_START;
      A(;
      L     "AI-SENSOR-DATA".JEN1_IC_SICAKLIK_ANLIK;
      L     "JEN1_DATA".SICAKLIK_SET_POINT_1;
      <R;
      );
      A(;
      L     "AI-SENSOR-DATA".JEN1_BASINC_ANLIK;
      L     "JEN1_DATA".BASINC_SET_POINT;
      <R;
      );
      O;
      A     "JEN1_DATA".OUT_BURLOR_MOT_START;
      AN    "JEN1_DATA".SICAKLIK_SET1_OK;
      );
      =     L 2.0;
      A     L 2.0;
      BLD   102;
      =     "JEN1_DATA".OUT_BURLOR_MOT_START;
      A     L 2.0;
      FP    M 754.1;
      R     #st_Set_100_Derece;
      A     L 2.0;
      L     S5T#500MS;
      SD    T 40;
      NOP   0;
      NOP   0;
      NOP   0;
      A     T 40;
      R     "JEN1_DATA".EKRAN_START;
      A     L 2.0;
      BLD   102;
      S     "JEN1_DATA".SISTEM_BASLADI;
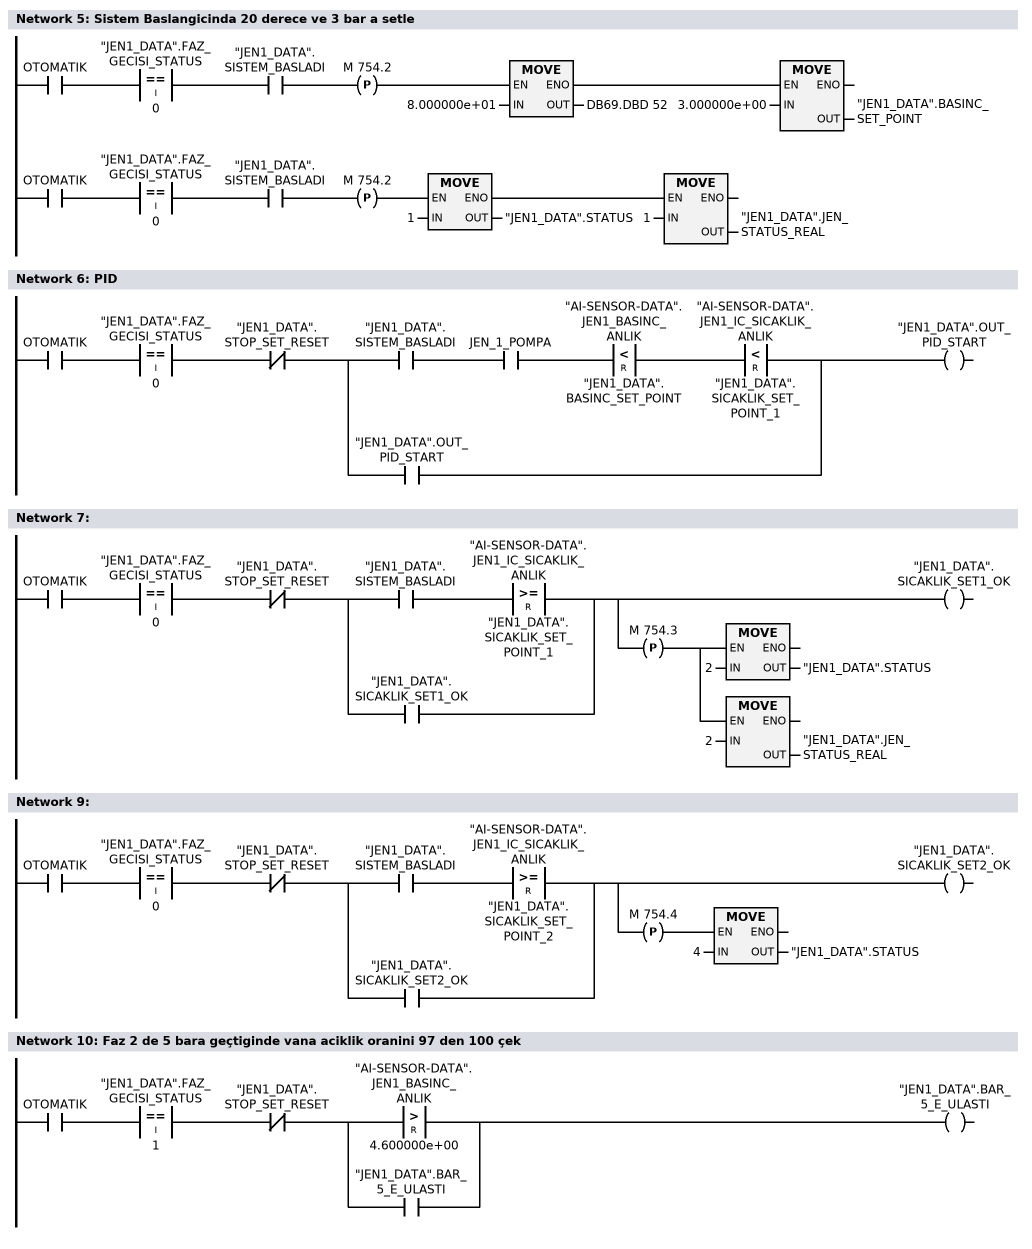
NETWORK
TITLE = Sistem Baslangicinda 20 derece ve 3 bar a setle
      A     "OTOMATIK";
      A(;
      L     "JEN1_DATA".FAZ_GECISI_STATUS;
      L     0;
      ==I;
      );
      A     "JEN1_DATA".SISTEM_BASLADI;
      FP    M 754.2;
      =     L 2.0;
      A(;
      A     L 2.0;
      JNB   _001;
      L     8.000000e+01;
      T     DB69.DBD 52;
      SET;
      SAVE;
      CLR;
_001: A     BR;
      );
      JNB   _002;
      L     3.000000e+00;
      T     "JEN1_DATA".BASINC_SET_POINT;
_002: NOP   0;
      A(;
      A     L 2.0;
      JNB   _003;
      L     1;
      T     "JEN1_DATA".STATUS;
      SET;
      SAVE;
      CLR;
_003: A     BR;
      );
      JNB   _004;
      L     1;
      T     "JEN1_DATA".JEN_STATUS_REAL;
_004: NOP   0;
NETWORK
TITLE = PID
      A     "OTOMATIK";
      A(;
      L     "JEN1_DATA".FAZ_GECISI_STATUS;
      L     0;
      ==I;
      );
      AN    "JEN1_DATA".STOP_SET_RESET;
      A(;
      A     "JEN1_DATA".SISTEM_BASLADI;
      A     "JEN_1_POMPA";
      A(;
      L     "AI-SENSOR-DATA".JEN1_BASINC_ANLIK;
      L     "JEN1_DATA".BASINC_SET_POINT;
      <R;
      );
      A(;
      L     "AI-SENSOR-DATA".JEN1_IC_SICAKLIK_ANLIK;
      L     "JEN1_DATA".SICAKLIK_SET_POINT_1;
      <R;
      );
      O     "JEN1_DATA".OUT_PID_START;
      );
      =     "JEN1_DATA".OUT_PID_START;
NETWORK
TITLE =
      A     "OTOMATIK";
      A(;
      L     "JEN1_DATA".FAZ_GECISI_STATUS;
      L     0;
      ==I;
      );
      AN    "JEN1_DATA".STOP_SET_RESET;
      A(;
      A     "JEN1_DATA".SISTEM_BASLADI;
      A(;
      L     "AI-SENSOR-DATA".JEN1_IC_SICAKLIK_ANLIK;
      L     "JEN1_DATA".SICAKLIK_SET_POINT_1;
      >=R;
      );
      O     "JEN1_DATA".SICAKLIK_SET1_OK;
      );
      =     L 2.0;
      A     L 2.0;
      BLD   102;
      =     "JEN1_DATA".SICAKLIK_SET1_OK;
      A     L 2.0;
      FP    M 754.3;
      =     L 2.1;
      A     L 2.1;
      JNB   _005;
      L     2;
      T     "JEN1_DATA".STATUS;
_005: NOP   0;
      A     L 2.1;
      JNB   _006;
      L     2;
      T     "JEN1_DATA".JEN_STATUS_REAL;
_006: NOP   0;
NETWORK
TITLE = SET 2 DEGERINE ULASMADI ISE BRULOR VE MOTORU CALISTIR
      A(;
      A     "JEN1_DATA".SICAKLIK_SET1_OK;
      FP    "SET2_ULASMADI_RIS";
      S     "SET2_ULASMADI_SR";
      A(;
      O(;
      L     "JEN1_DATA".FAZ_GECISI_STATUS;
      L     1;
      ==I;
      );
      O     "JEN1_DATA".STOP_SET_RESET;
      );
      R     "SET2_ULASMADI_SR";
      A     "SET2_ULASMADI_SR";
      );
      L     S5T#1M30S;
      SD    "TIM_SET2_ULASMADI";
      NOP   0;
      NOP   0;
      NOP   0;
      A     "TIM_SET2_ULASMADI";
      =     "JEN1_DATA".SET2_DEGERINE_ULASMADI;
NETWORK
TITLE =
      A     "OTOMATIK";
      A(;
      L     "JEN1_DATA".FAZ_GECISI_STATUS;
      L     0;
      ==I;
      );
      AN    "JEN1_DATA".STOP_SET_RESET;
      A(;
      A     "JEN1_DATA".SISTEM_BASLADI;
      A(;
      L     "AI-SENSOR-DATA".JEN1_IC_SICAKLIK_ANLIK;
      L     "JEN1_DATA".SICAKLIK_SET_POINT_2;
      >=R;
      );
      O     "JEN1_DATA".SICAKLIK_SET2_OK;
      );
      =     L 2.0;
      A     L 2.0;
      BLD   102;
      =     "JEN1_DATA".SICAKLIK_SET2_OK;
      A     L 2.0;
      FP    M 754.4;
      JNB   _007;
      L     4;
      T     "JEN1_DATA".STATUS;
_007: NOP   0;
NETWORK
TITLE = Faz 2 de 5 bara geçtiginde vana aciklik oranini 97 den 100 çek
      A     "OTOMATIK";
      A(;
      L     "JEN1_DATA".FAZ_GECISI_STATUS;
      L     1;
      ==I;
      );
      AN    "JEN1_DATA".STOP_SET_RESET;
      A(;
      O(;
      L     "AI-SENSOR-DATA".JEN1_BASINC_ANLIK;
      L     4.600000e+00;
      >R;
      );
      O     "JEN1_DATA".BAR_5_E_ULASTI;
      );
      =     "JEN1_DATA".BAR_5_E_ULASTI;
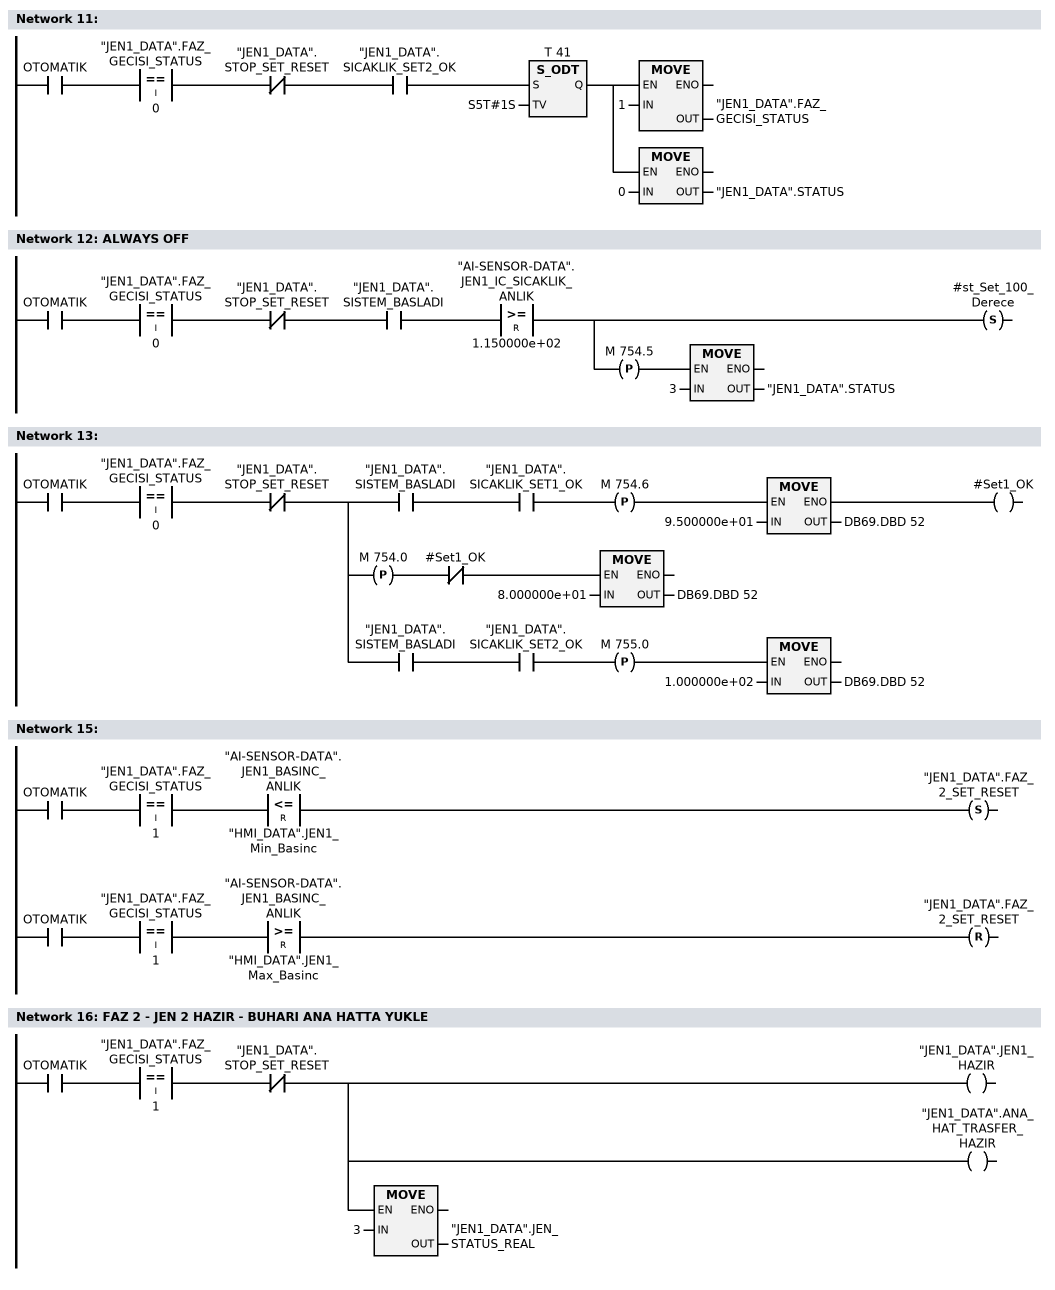
NETWORK
TITLE =
//SET 2 SICAKLIGINDAN SONRA FAZ 2 E GEC
      A     "OTOMATIK";
      A(;
      L     "JEN1_DATA".FAZ_GECISI_STATUS;
      L     0;
      ==I;
      );
      AN    "JEN1_DATA".STOP_SET_RESET;
      A     "JEN1_DATA".SICAKLIK_SET2_OK;
      L     S5T#1S;
      SD    T 41;
      NOP   0;
      NOP   0;
      NOP   0;
      A     T 41;
      =     L 2.0;
      A     L 2.0;
      JNB   _008;
      L     1;
      T     "JEN1_DATA".FAZ_GECISI_STATUS;
_008: NOP   0;
      A     L 2.0;
      JNB   _009;
      L     0;
      T     "JEN1_DATA".STATUS;
_009: NOP   0;
NETWORK
TITLE = ALWAYS OFF
//Pompa 100 derecede duracak
      A     "OTOMATIK";
      A(;
      L     "JEN1_DATA".FAZ_GECISI_STATUS;
      L     0;
      ==I;
      );
      AN    "JEN1_DATA".STOP_SET_RESET;
      A     "JEN1_DATA".SISTEM_BASLADI;
      A(;
      L     "AI-SENSOR-DATA".JEN1_IC_SICAKLIK_ANLIK;
      L     1.150000e+02;
      >=R;
      );
      =     L 2.0;
      A     L 2.0;
      BLD   102;
      S     #st_Set_100_Derece;
      A     L 2.0;
      FP    M 754.5;
      JNB   _00a;
      L     3;
      T     "JEN1_DATA".STATUS;
_00a: NOP   0;
NETWORK
TITLE =
//-Sicaklik set 1 e geldiginde vana kapanma orani 5'e kadar düsüyor
//-Sicaklik set 2 e geldiginde vana kapanma orani 0'a kadar dusecek
//
//m754.0
//
      A     "OTOMATIK";
      A(;
      L     "JEN1_DATA".FAZ_GECISI_STATUS;
      L     0;
      ==I;
      );
      AN    "JEN1_DATA".STOP_SET_RESET;
      =     L 2.0;
      A     L 2.0;
      A     "JEN1_DATA".SISTEM_BASLADI;
      A     "JEN1_DATA".SICAKLIK_SET1_OK;
      FP    M 754.6;
      JNB   _00b;
      L     9.500000e+01;
      T     DB69.DBD 52;
      SET;
      SAVE;
      CLR;
_00b: A     BR;
      =     #Set1_OK;
      A     L 2.0;
      FP    M 754.0;
      AN    #Set1_OK;
      JNB   _00c;
      L     8.000000e+01;
      T     DB69.DBD 52;
_00c: NOP   0;
      A     L 2.0;
      A     "JEN1_DATA".SISTEM_BASLADI;
      A     "JEN1_DATA".SICAKLIK_SET2_OK;
      FP    M 755.0;
      JNB   _00d;
      L     1.000000e+02;
      T     DB69.DBD 52;
_00d: NOP   0;
NETWORK
TITLE =
NETWORK
TITLE =
//FAZ - 2 MODUNA GEÇ
//1-BURLOR VE POMPA 4.5-5.5 BAR ARASINDA ÇALISIP DURACAK
      A     "OTOMATIK";
      A(;
      L     "JEN1_DATA".FAZ_GECISI_STATUS;
      L     1;
      ==I;
      );
      A(;
      L     "AI-SENSOR-DATA".JEN1_BASINC_ANLIK;
      L     "HMI_DATA".JEN1_Min_Basinc;
      <=R;
      );
      S     "JEN1_DATA".FAZ_2_SET_RESET;
      A     "OTOMATIK";
      A(;
      L     "JEN1_DATA".FAZ_GECISI_STATUS;
      L     1;
      ==I;
      );
      A(;
      L     "AI-SENSOR-DATA".JEN1_BASINC_ANLIK;
      L     "HMI_DATA".JEN1_Max_Basinc;
      >=R;
      );
      R     "JEN1_DATA".FAZ_2_SET_RESET;
      NOP   0;
NETWORK
TITLE = FAZ 2 - JEN 2 HAZIR - BUHARI ANA HATTA YUKLE
      A     "OTOMATIK";
      A(;
      L     "JEN1_DATA".FAZ_GECISI_STATUS;
      L     1;
      ==I;
      );
      AN    "JEN1_DATA".STOP_SET_RESET;
      =     L 2.0;
      A     L 2.0;
      BLD   102;
      =     "JEN1_DATA".JEN1_HAZIR;
      A     L 2.0;
      BLD   102;
      =     "JEN1_DATA".ANA_HAT_TRASFER_HAZIR;
      A     L 2.0;
      JNB   _00e;
      L     3;
      T     "JEN1_DATA".JEN_STATUS_REAL;
_00e: NOP   0;
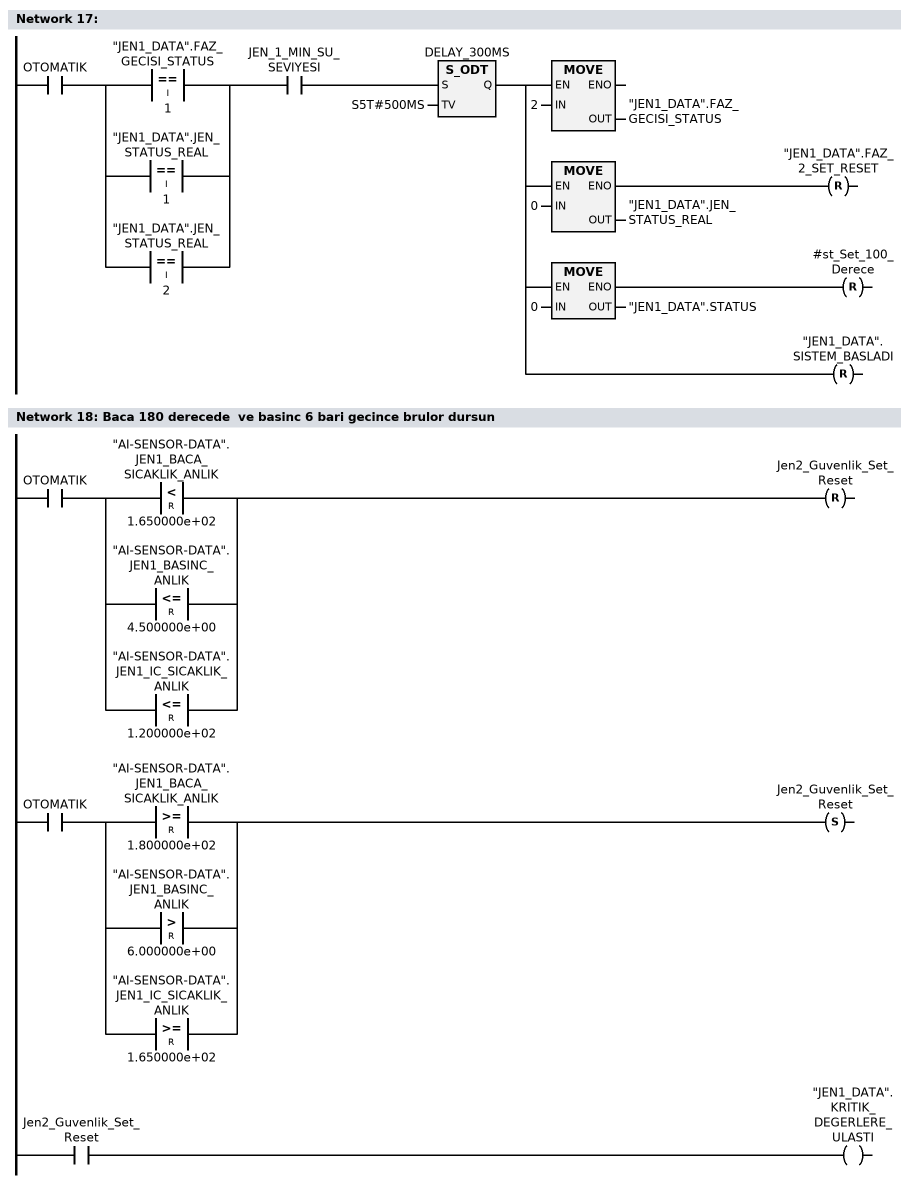
NETWORK
TITLE =
//FAZ 3 - GUVENLIK ONLEMLERI 
//1- 6 bar asildiginda -ok
//2- Baca 180 dereceyi gecerse -ok
//3- Su miktari min altina duserse -not ok
      A     "OTOMATIK";
      A(;
      O(;
      L     "JEN1_DATA".FAZ_GECISI_STATUS;
      L     1;
      ==I;
      );
      O(;
      L     "JEN1_DATA".JEN_STATUS_REAL;
      L     1;
      ==I;
      );
      O(;
      L     "JEN1_DATA".JEN_STATUS_REAL;
      L     2;
      ==I;
      );
      );
      A     "JEN_1_MIN_SU_SEVIYESI";
      L     S5T#500MS;
      SD    "DELAY_300MS";
      NOP   0;
      NOP   0;
      NOP   0;
      A     "DELAY_300MS";
      =     L 2.0;
      A     L 2.0;
      JNB   _00f;
      L     2;
      T     "JEN1_DATA".FAZ_GECISI_STATUS;
_00f: NOP   0;
      A     L 2.0;
      JNB   _010;
      L     0;
      T     "JEN1_DATA".JEN_STATUS_REAL;
      SET;
      SAVE;
      CLR;
_010: A     BR;
      R     "JEN1_DATA".FAZ_2_SET_RESET;
      A     L 2.0;
      JNB   _011;
      L     0;
      T     "JEN1_DATA".STATUS;
      SET;
      SAVE;
      CLR;
_011: A     BR;
      R     #st_Set_100_Derece;
      A     L 2.0;
      BLD   102;
      R     "JEN1_DATA".SISTEM_BASLADI;
NETWORK
TITLE = Baca 180 derecede  ve basinc 6 bari gecince brulor dursun
      A     "OTOMATIK";
      A(;
      O(;
      L     "AI-SENSOR-DATA".JEN1_BACA_SICAKLIK_ANLIK;
      L     1.650000e+02;
      <R;
      );
      O(;
      L     "AI-SENSOR-DATA".JEN1_BASINC_ANLIK;
      L     4.500000e+00;
      <=R;
      );
      O(;
      L     "AI-SENSOR-DATA".JEN1_IC_SICAKLIK_ANLIK;
      L     1.200000e+02;
      <=R;
      );
      );
      R     "Jen2_Guvenlik_Set_Reset";
      A     "OTOMATIK";
      A(;
      O(;
      L     "AI-SENSOR-DATA".JEN1_BACA_SICAKLIK_ANLIK;
      L     1.800000e+02;
      >=R;
      );
      O(;
      L     "AI-SENSOR-DATA".JEN1_BASINC_ANLIK;
      L     6.000000e+00;
      >R;
      );
      O(;
      L     "AI-SENSOR-DATA".JEN1_IC_SICAKLIK_ANLIK;
      L     1.650000e+02;
      >=R;
      );
      );
      S     "Jen2_Guvenlik_Set_Reset";
      A     "Jen2_Guvenlik_Set_Reset";
      =     "JEN1_DATA".KRITIK_DEGERLERE_ULASTI;
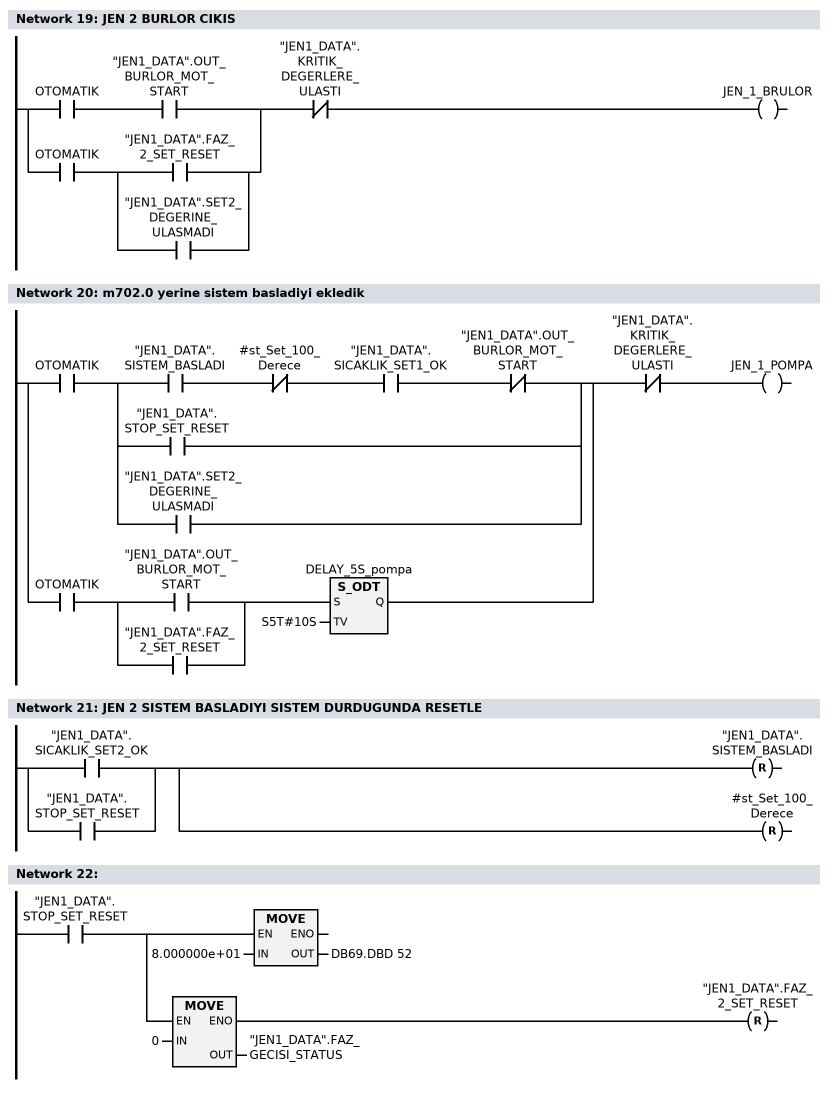
NETWORK
TITLE = JEN 2 BURLOR CIKIS
      A(;
      A     "OTOMATIK";
      A     "JEN1_DATA".OUT_BURLOR_MOT_START;
      O;
      A     "OTOMATIK";
      A(;
      O     "JEN1_DATA".FAZ_2_SET_RESET;
      O     "JEN1_DATA".SET2_DEGERINE_ULASMADI;
      );
      );
      AN    "JEN1_DATA".KRITIK_DEGERLERE_ULASTI;
      =     "JEN_1_BRULOR";
NETWORK
TITLE = m702.0 yerine sistem basladiyi ekledik
//q2.5 motor çikisi
      A(;
      A     "OTOMATIK";
      A(;
      A     "JEN1_DATA".SISTEM_BASLADI;
      AN    #st_Set_100_Derece;
      A     "JEN1_DATA".SICAKLIK_SET1_OK;
      AN    "JEN1_DATA".OUT_BURLOR_MOT_START;
      O     "JEN1_DATA".STOP_SET_RESET;
      O     "JEN1_DATA".SET2_DEGERINE_ULASMADI;
      );
      O(;
      A     "OTOMATIK";
      A(;
      O     "JEN1_DATA".OUT_BURLOR_MOT_START;
      O     "JEN1_DATA".FAZ_2_SET_RESET;
      );
      L     S5T#10S;
      SD    "DELAY_5S_pompa";
      NOP   0;
      NOP   0;
      NOP   0;
      A     "DELAY_5S_pompa";
      );
      );
      AN    "JEN1_DATA".KRITIK_DEGERLERE_ULASTI;
      =     "JEN_1_POMPA";
NETWORK
TITLE = JEN 2 SISTEM BASLADIYI SISTEM DURDUGUNDA RESETLE
      O     "JEN1_DATA".SICAKLIK_SET2_OK;
      O     "JEN1_DATA".STOP_SET_RESET;
      R     "JEN1_DATA".SISTEM_BASLADI;
      R     #st_Set_100_Derece;
NETWORK
TITLE =
      A     "JEN1_DATA".STOP_SET_RESET;
      =     L 2.0;
      A     L 2.0;
      JNB   _012;
      L     8.000000e+01;
      T     DB69.DBD 52;
_012: NOP   0;
      A     L 2.0;
      JNB   _013;
      L     0;
      T     "JEN1_DATA".FAZ_GECISI_STATUS;
      SET;
      SAVE;
      CLR;
_013: A     BR;
      R     "JEN1_DATA".FAZ_2_SET_RESET;
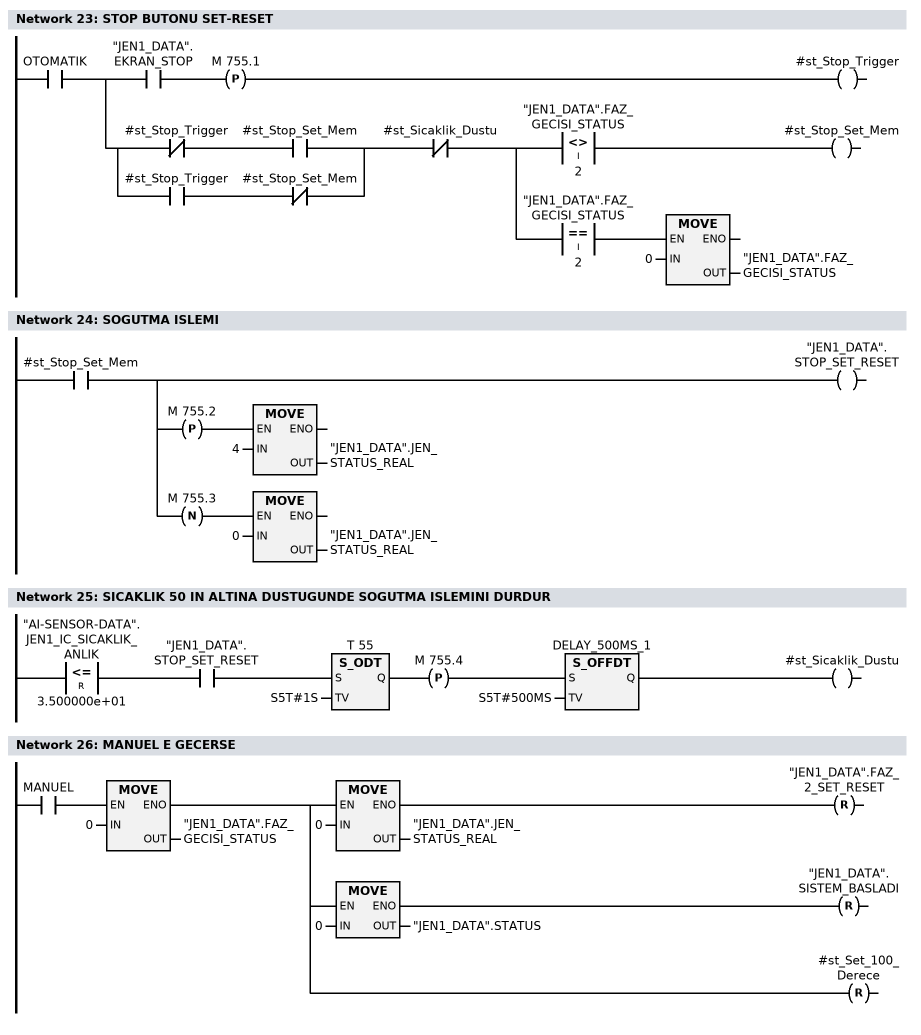
NETWORK
TITLE = STOP BUTONU SET-RESET
      A     "OTOMATIK";
      =     L 2.0;
      A     L 2.0;
      A     "JEN1_DATA".EKRAN_STOP;
      FP    M 755.1;
      =     #st_Stop_Trigger;
      A     L 2.0;
      A(;
      AN    #st_Stop_Trigger;
      A     #st_Stop_Set_Mem;
      O;
      A     #st_Stop_Trigger;
      AN    #st_Stop_Set_Mem;
      );
      AN    #st_Sicaklik_Dustu;
      =     L 2.1;
      A     L 2.1;
      A(;
      L     "JEN1_DATA".FAZ_GECISI_STATUS;
      L     2;
      <>I;
      );
      =     #st_Stop_Set_Mem;
      A     L 2.1;
      A(;
      L     "JEN1_DATA".FAZ_GECISI_STATUS;
      L     2;
      ==I;
      );
      JNB   _014;
      L     0;
      T     "JEN1_DATA".FAZ_GECISI_STATUS;
_014: NOP   0;
NETWORK
TITLE = SOGUTMA ISLEMI
      A     #st_Stop_Set_Mem;
      =     L 2.0;
      A     L 2.0;
      BLD   102;
      =     "JEN1_DATA".STOP_SET_RESET;
      A     L 2.0;
      FP    M 755.2;
      JNB   _015;
      L     4;
      T     "JEN1_DATA".JEN_STATUS_REAL;
_015: NOP   0;
      A     L 2.0;
      FN    M 755.3;
      JNB   _016;
      L     0;
      T     "JEN1_DATA".JEN_STATUS_REAL;
_016: NOP   0;
NETWORK
TITLE = SICAKLIK 50 IN ALTINA DUSTUGUNDE SOGUTMA ISLEMINI DURDUR
      A(;
      A(;
      L     "AI-SENSOR-DATA".JEN1_IC_SICAKLIK_ANLIK;
      L     3.500000e+01;
      <=R;
      );
      A     "JEN1_DATA".STOP_SET_RESET;
      L     S5T#1S;
      SD    T 55;
      NOP   0;
      NOP   0;
      NOP   0;
      A     T 55;
      );
      FP    M 755.4;
      L     S5T#500MS;
      SF    "DELAY_500MS_1";
      NOP   0;
      NOP   0;
      NOP   0;
      A     "DELAY_500MS_1";
      =     #st_Sicaklik_Dustu;
NETWORK
TITLE = MANUEL E GECERSE
      A     "MANUEL";
      JNB   _017;
      L     0;
      T     "JEN1_DATA".FAZ_GECISI_STATUS;
      SET;
      SAVE;
      CLR;
_017: A     BR;
      =     L 2.0;
      A     L 2.0;
      JNB   _018;
      L     0;
      T     "JEN1_DATA".JEN_STATUS_REAL;
      SET;
      SAVE;
      CLR;
_018: A     BR;
      R     "JEN1_DATA".FAZ_2_SET_RESET;
      A     L 2.0;
      JNB   _019;
      L     0;
      T     "JEN1_DATA".STATUS;
      SET;
      SAVE;
      CLR;
_019: A     BR;
      R     "JEN1_DATA".SISTEM_BASLADI;
      A     L 2.0;
      BLD   102;
      R     #st_Set_100_Derece;
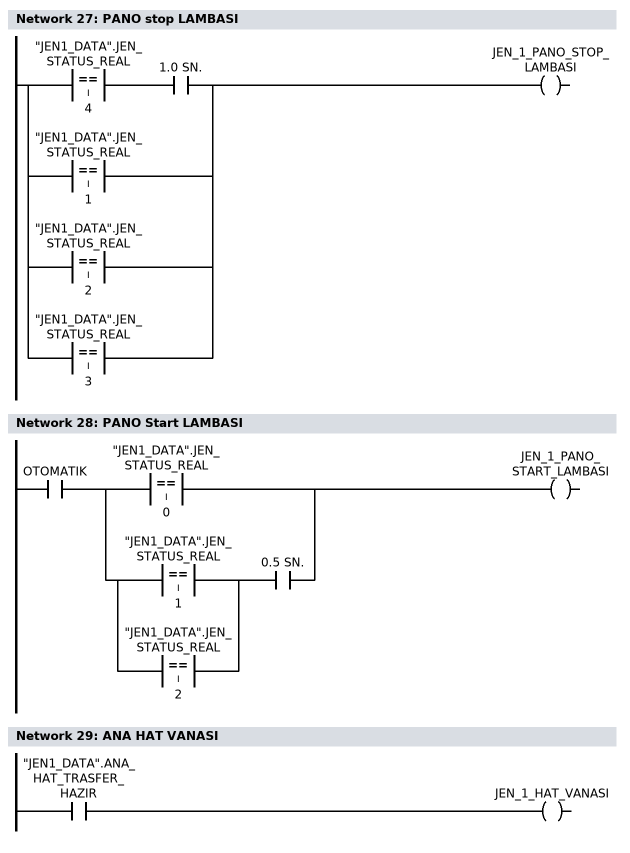
NETWORK
TITLE = PANO stop LAMBASI
      A(;
      L     "JEN1_DATA".JEN_STATUS_REAL;
      L     4;
      ==I;
      );
      A     "1.0 SN.";
      O(;
      L     "JEN1_DATA".JEN_STATUS_REAL;
      L     1;
      ==I;
      );
      O(;
      L     "JEN1_DATA".JEN_STATUS_REAL;
      L     2;
      ==I;
      );
      O(;
      L     "JEN1_DATA".JEN_STATUS_REAL;
      L     3;
      ==I;
      );
      =     "JEN_1_PANO_STOP_LAMBASI";
NETWORK
TITLE = PANO Start LAMBASI
      A     "OTOMATIK";
      A(;
      O(;
      L     "JEN1_DATA".JEN_STATUS_REAL;
      L     0;
      ==I;
      );
      O;
      A(;
      O(;
      L     "JEN1_DATA".JEN_STATUS_REAL;
      L     1;
      ==I;
      );
      O(;
      L     "JEN1_DATA".JEN_STATUS_REAL;
      L     2;
      ==I;
      );
      );
      A     "0.5 SN.";
      );
      =     "JEN_1_PANO_START_LAMBASI";
NETWORK
TITLE = ANA HAT VANASI 
      A     "JEN1_DATA".ANA_HAT_TRASFER_HAZIR;
      =     "JEN_1_HAT_VANASI";
END_FUNCTION_BLOCK

FUNCTION_BLOCK "JEN2_KONTROL_BLOGU"	// FB 99
//PIW 286 - Jen 2 Basinc
//PIW 288 - Jen 2 Buhar Sicakligi
//PQW 278 - Jen 2 Baca Sicakligi
VERSION : 0.1
VAR
  Rising_Status : BOOL ;
  Rising_Startup : BOOL ;
  Set_100_Derece : BOOL ;
  Rising_After_Stop : BOOL ;
  Set1_OK : BOOL ;
  Rising_Status_3 : BOOL ;
  Rising_Status_4 : BOOL ;
  Rising_100_dere_reset : BOOL ;
  Ris_Set1_ok_95 : BOOL ;
  Ris_Set2_ok_100 : BOOL ;
END_VAR
BEGIN
NETWORK
TITLE = Analog Çeviriler
      A     "ALWAYS OFF";
      =     L 0.0;
      BLD   103;
      A(;
      A     "ALWAYS OFF";
      =     L 0.1;
      BLD   103;
      CALL  "SCALE" (
           $1                       := P#P 286.0,
           $2                       := L#1092616192,
           $3                       := L#0,
           $4                       := L 0.1,
           $5                       := "AI-SENSOR-DATA".JEN2_BASINC_RET_VAL,
           $6                       := "AI-SENSOR-DATA".JEN2_BASINC_ANLIK);
      A     BR;
      );
      JNB   _001;
      CALL  "SCALE" (
           $1                       := P#P 288.0,
           $2                       := L#1128792064,
           $3                       := L#0,
           $4                       := L 0.0,
           $5                       := "AI-SENSOR-DATA".JEN2_IC_SICAKLIK_RET_VAL,
           $6                       := "AI-SENSOR-DATA".JEN2_IC_SICAKLIK_ANLIK);
_001: NOP   0;
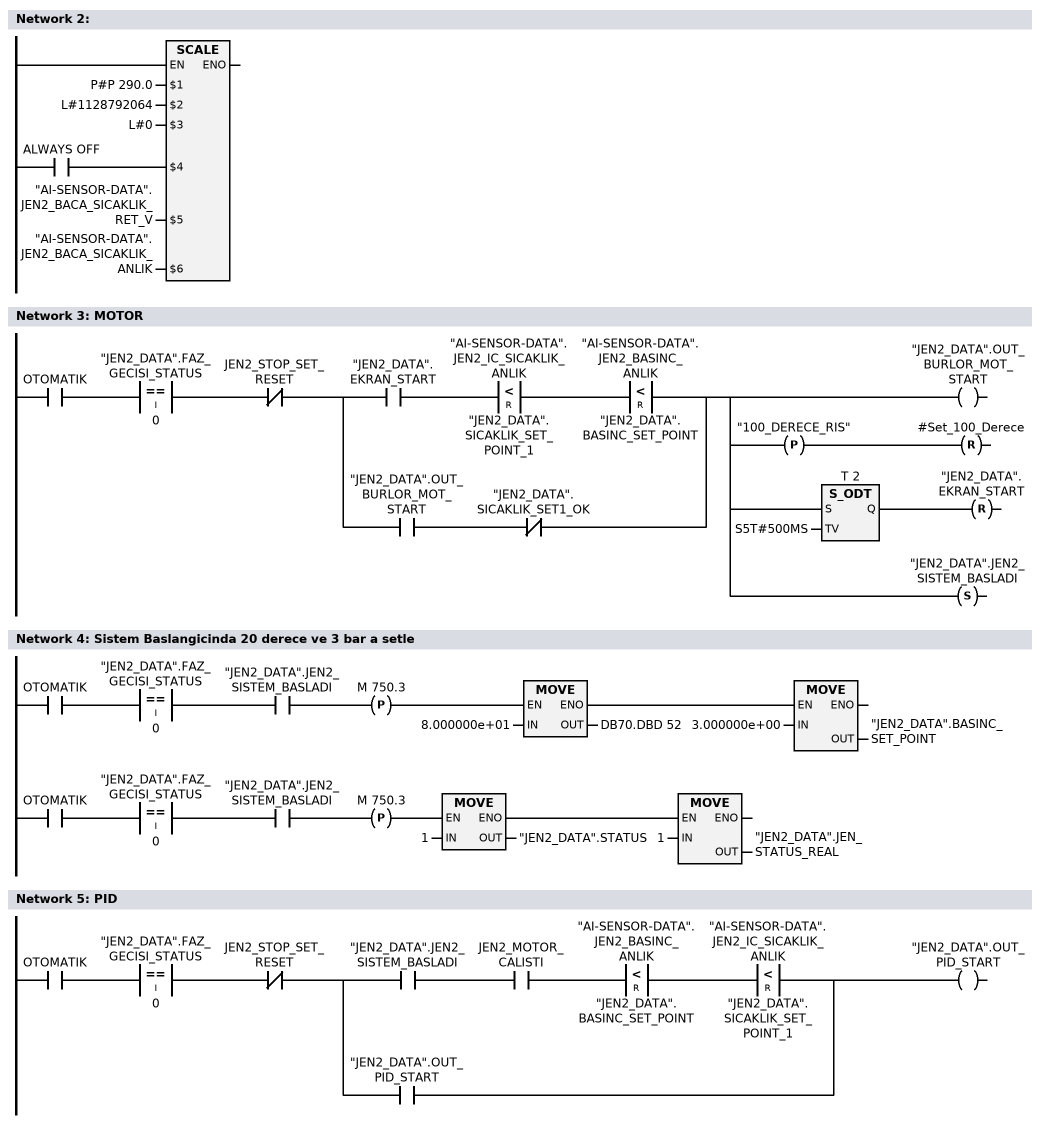
NETWORK
TITLE =
      A     "ALWAYS OFF";
      =     L 0.0;
      BLD   103;
      CALL  "SCALE" (
           $1                       := P#P 290.0,
           $2                       := L#1128792064,
           $3                       := L#0,
           $4                       := L 0.0,
           $5                       := "AI-SENSOR-DATA".JEN2_BACA_SICAKLIK_RET_V,
           $6                       := "AI-SENSOR-DATA".JEN2_BACA_SICAKLIK_ANLIK);
      NOP   0;
NETWORK
TITLE = MOTOR
      A     "OTOMATIK";
      A(;
      L     "JEN2_DATA".FAZ_GECISI_STATUS;
      L     0;
      ==I;
      );
      AN    "JEN2_STOP_SET_RESET";
      A(;
      A     "JEN2_DATA".EKRAN_START;
      A(;
      L     "AI-SENSOR-DATA".JEN2_IC_SICAKLIK_ANLIK;
      L     "JEN2_DATA".SICAKLIK_SET_POINT_1;
      <R;
      );
      A(;
      L     "AI-SENSOR-DATA".JEN2_BASINC_ANLIK;
      L     "JEN2_DATA".BASINC_SET_POINT;
      <R;
      );
      O;
      A     "JEN2_DATA".OUT_BURLOR_MOT_START;
      AN    "JEN2_DATA".SICAKLIK_SET1_OK;
      );
      =     L 0.0;
      A     L 0.0;
      BLD   102;
      =     "JEN2_DATA".OUT_BURLOR_MOT_START;
      A     L 0.0;
      FP    "100_DERECE_RIS";
      R     #Set_100_Derece;
      A     L 0.0;
      L     S5T#500MS;
      SD    T 2;
      NOP   0;
      NOP   0;
      NOP   0;
      A     T 2;
      R     "JEN2_DATA".EKRAN_START;
      A     L 0.0;
      BLD   102;
      S     "JEN2_DATA".JEN2_SISTEM_BASLADI;
NETWORK
TITLE = Sistem Baslangicinda 20 derece ve 3 bar a setle
      A     "OTOMATIK";
      A(;
      L     "JEN2_DATA".FAZ_GECISI_STATUS;
      L     0;
      ==I;
      );
      A     "JEN2_DATA".JEN2_SISTEM_BASLADI;
      FP    M 750.3;
      =     L 0.0;
      A(;
      A     L 0.0;
      JNB   _002;
      L     8.000000e+01;
      T     DB70.DBD 52;
      SET;
      SAVE;
      CLR;
_002: A     BR;
      );
      JNB   _003;
      L     3.000000e+00;
      T     "JEN2_DATA".BASINC_SET_POINT;
_003: NOP   0;
      A(;
      A     L 0.0;
      JNB   _004;
      L     1;
      T     "JEN2_DATA".STATUS;
      SET;
      SAVE;
      CLR;
_004: A     BR;
      );
      JNB   _005;
      L     1;
      T     "JEN2_DATA".JEN_STATUS_REAL;
_005: NOP   0;
NETWORK
TITLE = PID
      A     "OTOMATIK";
      A(;
      L     "JEN2_DATA".FAZ_GECISI_STATUS;
      L     0;
      ==I;
      );
      AN    "JEN2_STOP_SET_RESET";
      A(;
      A     "JEN2_DATA".JEN2_SISTEM_BASLADI;
      A     "JEN2_MOTOR_CALISTI";
      A(;
      L     "AI-SENSOR-DATA".JEN2_BASINC_ANLIK;
      L     "JEN2_DATA".BASINC_SET_POINT;
      <R;
      );
      A(;
      L     "AI-SENSOR-DATA".JEN2_IC_SICAKLIK_ANLIK;
      L     "JEN2_DATA".SICAKLIK_SET_POINT_1;
      <R;
      );
      O     "JEN2_DATA".OUT_PID_START;
      );
      =     "JEN2_DATA".OUT_PID_START;
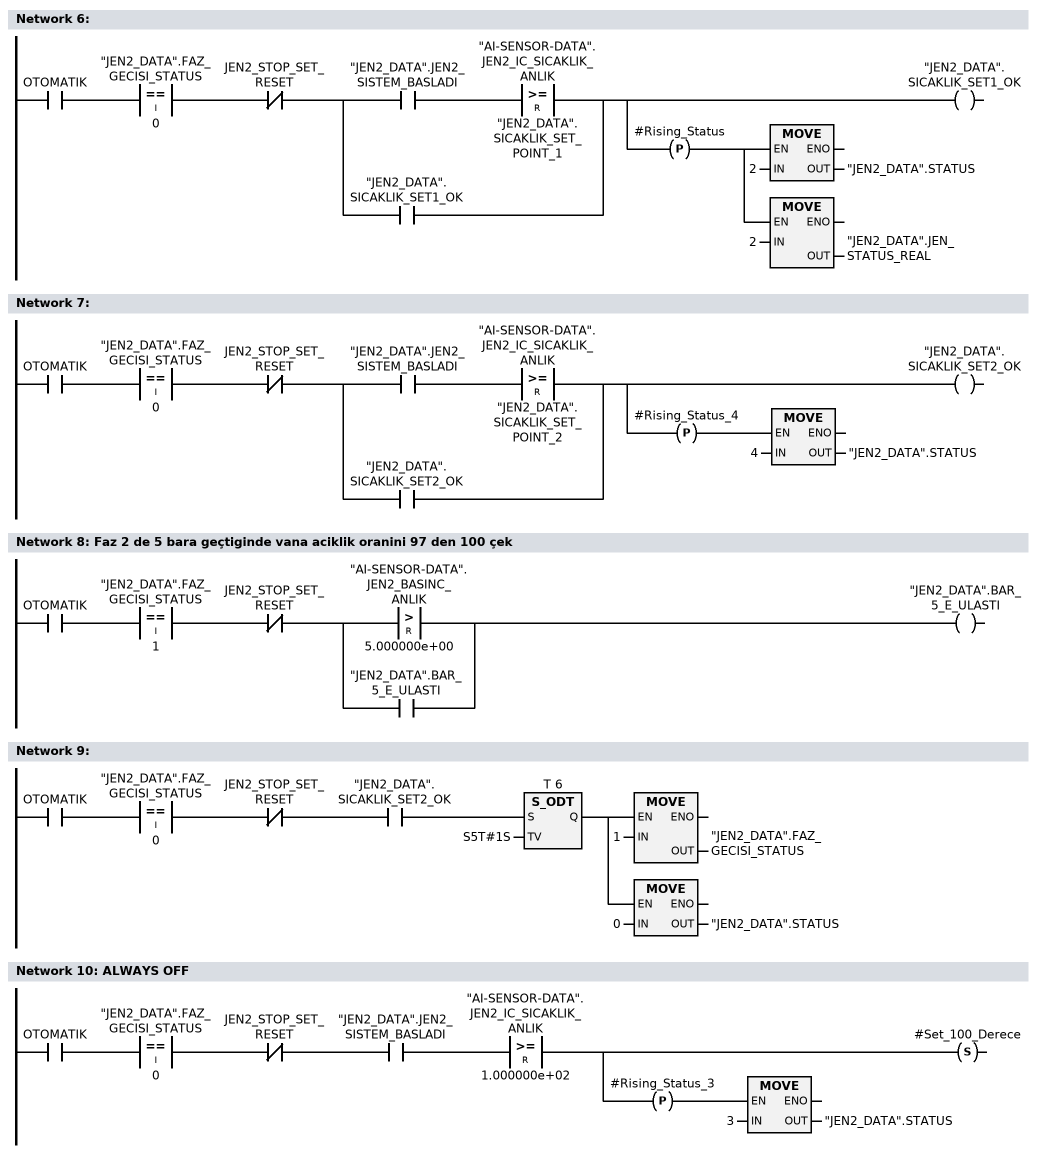
NETWORK
TITLE =
      A     "OTOMATIK";
      A(;
      L     "JEN2_DATA".FAZ_GECISI_STATUS;
      L     0;
      ==I;
      );
      AN    "JEN2_STOP_SET_RESET";
      A(;
      A     "JEN2_DATA".JEN2_SISTEM_BASLADI;
      A(;
      L     "AI-SENSOR-DATA".JEN2_IC_SICAKLIK_ANLIK;
      L     "JEN2_DATA".SICAKLIK_SET_POINT_1;
      >=R;
      );
      O     "JEN2_DATA".SICAKLIK_SET1_OK;
      );
      =     L 0.0;
      A     L 0.0;
      BLD   102;
      =     "JEN2_DATA".SICAKLIK_SET1_OK;
      A     L 0.0;
      FP    #Rising_Status;
      =     L 0.1;
      A     L 0.1;
      JNB   _006;
      L     2;
      T     "JEN2_DATA".STATUS;
_006: NOP   0;
      A     L 0.1;
      JNB   _007;
      L     2;
      T     "JEN2_DATA".JEN_STATUS_REAL;
_007: NOP   0;
NETWORK
TITLE =
      A     "OTOMATIK";
      A(;
      L     "JEN2_DATA".FAZ_GECISI_STATUS;
      L     0;
      ==I;
      );
      AN    "JEN2_STOP_SET_RESET";
      A(;
      A     "JEN2_DATA".JEN2_SISTEM_BASLADI;
      A(;
      L     "AI-SENSOR-DATA".JEN2_IC_SICAKLIK_ANLIK;
      L     "JEN2_DATA".SICAKLIK_SET_POINT_2;
      >=R;
      );
      O     "JEN2_DATA".SICAKLIK_SET2_OK;
      );
      =     L 0.0;
      A     L 0.0;
      BLD   102;
      =     "JEN2_DATA".SICAKLIK_SET2_OK;
      A     L 0.0;
      FP    #Rising_Status_4;
      JNB   _008;
      L     4;
      T     "JEN2_DATA".STATUS;
_008: NOP   0;
NETWORK
TITLE = Faz 2 de 5 bara geçtiginde vana aciklik oranini 97 den 100 çek
      A     "OTOMATIK";
      A(;
      L     "JEN2_DATA".FAZ_GECISI_STATUS;
      L     1;
      ==I;
      );
      AN    "JEN2_STOP_SET_RESET";
      A(;
      O(;
      L     "AI-SENSOR-DATA".JEN2_BASINC_ANLIK;
      L     5.000000e+00;
      >R;
      );
      O     "JEN2_DATA".BAR_5_E_ULASTI;
      );
      =     "JEN2_DATA".BAR_5_E_ULASTI;
NETWORK
TITLE =
//SET 2 SICAKLIGINDAN SONRA FAZ 2 E GEC
      A     "OTOMATIK";
      A(;
      L     "JEN2_DATA".FAZ_GECISI_STATUS;
      L     0;
      ==I;
      );
      AN    "JEN2_STOP_SET_RESET";
      A     "JEN2_DATA".SICAKLIK_SET2_OK;
      L     S5T#1S;
      SD    T 6;
      NOP   0;
      NOP   0;
      NOP   0;
      A     T 6;
      =     L 0.0;
      A     L 0.0;
      JNB   _009;
      L     1;
      T     "JEN2_DATA".FAZ_GECISI_STATUS;
_009: NOP   0;
      A     L 0.0;
      JNB   _00a;
      L     0;
      T     "JEN2_DATA".STATUS;
_00a: NOP   0;
NETWORK
TITLE = ALWAYS OFF
//Pompa 100 derecede duracak
      A     "OTOMATIK";
      A(;
      L     "JEN2_DATA".FAZ_GECISI_STATUS;
      L     0;
      ==I;
      );
      AN    "JEN2_STOP_SET_RESET";
      A     "JEN2_DATA".JEN2_SISTEM_BASLADI;
      A(;
      L     "AI-SENSOR-DATA".JEN2_IC_SICAKLIK_ANLIK;
      L     1.000000e+02;
      >=R;
      );
      =     L 0.0;
      A     L 0.0;
      BLD   102;
      S     #Set_100_Derece;
      A     L 0.0;
      FP    #Rising_Status_3;
      JNB   _00b;
      L     3;
      T     "JEN2_DATA".STATUS;
_00b: NOP   0;
